# B&R Automation Studio project Parker_BMM_ST_V5_3147_V12 (part 14)

#### robot.c
```c
/********************************************************************
 * COPYRIGHT --  B&R
 ********************************************************************
 * Program: robot
 * File: robot.c
 * Author: lijianjun
 * Created: March 06, 2013
 ********************************************************************
 * Implementation of program robot --- robot control
 ********************************************************************/

#include <bur/plctypes.h>

#ifdef _DEFAULT_INCLUDES
#include <AsDefault.h>
#endif

/**************************************************************************************
                            Function Declarations
**************************************************************************************/
void RobotTransfer( Mold_typ * pMold,Robot_Para_typ * pRobotPara, Robot_Transfer_Fix_typ * pRobotTransferFix, Robot_UpDn_Fix_typ * pRobotUpDnFix );
void RobotTransfer_Drive( Mold_typ * pMold,Robot_Para_typ * pRobotPara, Robot_Transfer_Fix_typ * pRobotTransferFix, Robot_UpDn_Fix_typ * pRobotUpDnFix );

/**************************************************************************************
     	        		I N I T U P  O F   T H E   T A S K
**************************************************************************************/
_INIT void init ( void )
{
	RTInfo_Task.enable = 1;
	RTInfo(&RTInfo_Task);

	tTask = RTInfo_Task.cycle_time/1000.0/1000.0;		/*  from us ---> s  */

	LMold.Robot.Step = 30000;
	RMold.Robot.Step = 30000;

} /* end of _INIT */

 /*************************************************************************************
        				C Y C L I C   P A R T   O F   T H E   T A S K
**************************************************************************************/

_CYCLIC void cyclic ( void )
{
	if(LMold.TimeSet.RobotFwAlarmTime  == 0)LMold.TimeSet.RobotFwAlarmTime = 1000;	/*  10s  */
	if(LMold.TimeSet.RobotBwAlarmTime  == 0)LMold.TimeSet.RobotBwAlarmTime = 1000;
	if(LMold.TimeSet.RobotUpAlarmTime  == 0)LMold.TimeSet.RobotUpAlarmTime = 1000;
	if(LMold.TimeSet.RobotDnAlarmTime  == 0)LMold.TimeSet.RobotDnAlarmTime = 1000;

	if(RMold.TimeSet.RobotFwAlarmTime  == 0)RMold.TimeSet.RobotFwAlarmTime = 1000;	/*  10s  */
	if(RMold.TimeSet.RobotBwAlarmTime  == 0)RMold.TimeSet.RobotBwAlarmTime = 1000;
	if(RMold.TimeSet.RobotUpAlarmTime  == 0)RMold.TimeSet.RobotUpAlarmTime = 1000;
	if(RMold.TimeSet.RobotDnAlarmTime  == 0)RMold.TimeSet.RobotDnAlarmTime = 1000;

	LMold.TransDIn.RobotBwLimit = gMachineIn.LMold.RobotBwLimit;
	RMold.TransDIn.RobotBwLimit = gMachineIn.RMold.RobotBwLimit;

	LMold.TransDIn.RobotFwLimit = gMachineIn.LMold.RobotFwLimit;
	RMold.TransDIn.RobotFwLimit = gMachineIn.RMold.RobotFwLimit;

	LMold.TransDIn.RobotFwSlowLimit = gMachineIn.LMold.RobotFwSlowLimit;
	RMold.TransDIn.RobotFwSlowLimit = gMachineIn.RMold.RobotFwSlowLimit;

	LMold.TransDIn.RobotUpLimit = gMachineIn.LMold.RobotUpLimit;
	LMold.TransDIn.RobotDnLimit = gMachineIn.LMold.RobotDnLimit;

	RMold.TransDIn.RobotUpLimit = gMachineIn.RMold.RobotUpLimit;
	RMold.TransDIn.RobotDnLimit = gMachineIn.RMold.RobotDnLimit;

	//Ext Robot
	LMold.TransDIn.ExtRobotUpLmit = gMachineIn.LMold.ExtRobotUpLimit;
	RMold.TransDIn.ExtRobotUpLmit = gMachineIn.RMold.ExtRobotUpLimit;

	if(ACTUATOR_ELECTRIC == gMachineFix.MoldR.RobotTransfer.eActuatorType)
	{
		if(0 == gMachineFix.Option.bHideLeftStation)  // two mold
		{
			RobotTransfer_Drive(&LMold,&gMachinePara.MoldL.Robot,&gMachineFix.MoldL.RobotTransfer,&gMachineFix.MoldL.RobotUpDn);
		}
		RobotTransfer_Drive(&RMold,&gMachinePara.MoldR.Robot,&gMachineFix.MoldR.RobotTransfer,&gMachineFix.MoldR.RobotUpDn);
	}
	else
	{
		if(0 == gMachineFix.Option.bHideLeftStation)  // two mold
		{
			RobotTransfer(&LMold,&gMachinePara.MoldL.Robot,&gMachineFix.MoldL.RobotTransfer,&gMachineFix.MoldL.RobotUpDn);
		}
		RobotTransfer(&RMold,&gMachinePara.MoldR.Robot,&gMachineFix.MoldR.RobotTransfer,&gMachineFix.MoldR.RobotUpDn);
	}

	gMachineOut.LMold.RobotFw = LMold.ValveOut.RobotFw;
	gMachineOut.LMold.RobotBw = LMold.ValveOut.RobotBw;

	gMachineOut.RMold.RobotFw = RMold.ValveOut.RobotFw;
	gMachineOut.RMold.RobotBw = RMold.ValveOut.RobotBw;

	gMachineOut.LMold.RobotUp = LMold.ValveOut.RobotUp;
	gMachineOut.LMold.RobotDn = LMold.ValveOut.RobotDn;

	gMachineOut.RMold.RobotUp = RMold.ValveOut.RobotUp;
	gMachineOut.RMold.RobotDn = RMold.ValveOut.RobotDn;

	//		gMachineOut.LMold.ProductAuxClamp = LMold.ValveOut.ProductAuxClamp;
	//		gMachineOut.RMold.ProductAuxClamp = RMold.ValveOut.ProductAuxClamp;

	/*---------------------------------------------------*/
	/*----------------- Robot Transfer-----------------*/
	/*------------- ActuatorType--------------- */
	gMachineFix.MoldL.RobotTransfer.eActuatorType = gMachineFix.MoldR.RobotTransfer.eActuatorType;

	/*-------------- ValveType----------------- */
	gMachineFix.MoldL.RobotTransfer.eValveType = gMachineFix.MoldR.RobotTransfer.eValveType;

	/*------------ PressueOutputType--------------- */
	gMachineFix.MoldL.RobotTransfer.ePressueOutputType = gMachineFix.MoldR.RobotTransfer.ePressueOutputType;

	/*------------ FluxOutputType--------------- */
	gMachineFix.MoldL.RobotTransfer.eFluxOutputType = gMachineFix.MoldR.RobotTransfer.eFluxOutputType;

	/*---------------------------------------------------*/
	/*----------------- Robot UpDn-----------------*/
	/*------------- ActuatorType--------------- */
	gMachineFix.MoldL.RobotUpDn.eActuatorType = gMachineFix.MoldR.RobotUpDn.eActuatorType;

	/*-------------- ValveType----------------- */
	gMachineFix.MoldL.RobotUpDn.eValveType = gMachineFix.MoldR.RobotUpDn.eValveType;

	/*------------ PressueOutputType--------------- */
	gMachineFix.MoldL.RobotUpDn.ePressueOutputType = gMachineFix.MoldR.RobotUpDn.ePressueOutputType;

	/*------------ FluxOutputType--------------- */
	gMachineFix.MoldL.RobotUpDn.eFluxOutputType = gMachineFix.MoldR.RobotUpDn.eFluxOutputType;

	/*---------------Motor Trand-------------*/
	gMotorTrace.RMold.RobotTransfer.Position 		= RMold.Robot.Transfer.mmAs;

} /* end of _CYCLIC */

void RobotTransfer( Mold_typ * pMold,Robot_Para_typ * pRobotPara, Robot_Transfer_Fix_typ * pRobotTransferFix, Robot_UpDn_Fix_typ * pRobotUpDnFix )
{
	if(pMold == & LMold)
	{
		pRobotTransferFix->pMax = gMachineFix.Pump.MaxP2;
	}
	else
	{
		pRobotTransferFix->pMax = gMachineFix.Pump.MaxP1;
	}

	pMold->Robot.Transfer.FwPos = pMold->TransDIn.RobotFwLimit;
	pMold->Robot.Transfer.BwPos = pMold->TransDIn.RobotBwLimit;

	pMold->Robot.UpDn.UpPos = pMold->TransDIn.RobotUpLimit;
	pMold->Robot.UpDn.DnPos = pMold->TransDIn.RobotDnLimit;

	switch ( pMold->Robot.Step )
	{
		/*------------------ stop all the output ------------------*/
		case 0:

			switch (pRobotTransferFix->eActuatorType)
			{
				/*-------------------------------------------------*/
				case ACTUATOR_HYD: /*1:Oil*/
					/*-------------------------------------------------*/

					pMold->ActInfo.RobotFw	= 0;
					pMold->ActInfo.RobotBw	= 0;

					pMold->ValveOut.RobotFw = 0;
					pMold->ValveOut.RobotBw = 0;

					pMold->Robot.Transfer.p_set = 0;
					pMold->Robot.Transfer.v_set = 0;
					break;
				/*-------------------------------------------------*/
				case ACTUATOR_PNEU: /*2:Air*/
					/*-------------------------------------------------*/

					break;
			}

			pMold->Robot.Timer.IN = 0;
			pMold->Robot.LimitTimer.IN = 0;

			break;

		/*--------------------------------------------------- */
		/*------------------ Robot Fw ----------------------- */
		/*--------------------------------------------------- */
		case 100:		/* Fw delay */
			if(1 == pMold->Option.RobotTransfer)
			{
				if(pMold->TimeSet.RobotFwDly != 0)
				{
					pMold->Robot.Timer.IN = 1;
					pMold->Robot.Timer.PT = pMold->TimeSet.RobotFwDly;

					if(1 == gMachineInfo.Auto)
					{
						if(13000 == pMold->RobotOpnCls.Step || 0 == pMold->RobotOpnCls.Step)  // Opn too Slow wait, Opn Done
						{
							pMold->Robot.Step = 200;
						}
					}
					else
					{
						pMold->Robot.Step = 200;
					}
				}
				else
				{
					if(1 == gMachineInfo.Auto)
					{
						if(13000 == pMold->RobotOpnCls.Step || 0 == pMold->RobotOpnCls.Step)  // Opn too Slow wait, Opn Done
						{
							pMold->Robot.Step = 300;
						}
					}
					else
					{
						pMold->Robot.Step = 300;
					}
				}
			}
			else
			{
				pMold->Robot.Step = 300;
			}

			break;

		case 200:  		/* delay ok */
			pMold->TimeDis.RobotFwDly = pMold->Robot.Timer.ET;
			if (1 == pMold->Robot.Timer.Q)
			{
				pMold->Robot.Timer.IN        = 0;
				pMold->Robot.Step = 300;
			}
			break;

		case 300:  		/* set time */

			if(1 == pMold->Option.RobotTransfer)
			{
				pMold->Robot.LimitTimer.IN = 1;
				pMold->Robot.LimitTimer.PT = pMold->TimeSet.RobotFwAlarmTime;

				pMold->Robot.Step = 400;
			}
			else
			{
				pMold->Robot.Step = 2900; // for no use
			}
			break;

		case 400: // Fw quick
			pMold->ActInfo.RobotFw  = 1;
			pMold->ActInfo.RobotBw  = 0;

			switch (pRobotTransferFix->eActuatorType)
			{
				/*-------------------------------------------------*/
				case ACTUATOR_HYD: /*1:Oil*/
					/*-------------------------------------------------*/
					pMold->ValveOut.RobotFw = 1;
					pMold->ValveOut.RobotBw = 0;

					pMold->Robot.Transfer.p_set = pRobotPara->ParaTransfer.P_Fw;
					pMold->Robot.Transfer.v_set = pRobotPara->ParaTransfer.V_Fw;

					if(1 == pMold->TransDIn.RobotFwLimit || 1 == pMold->TransDIn.RobotFwSlowLimit)
					{
						pMold->Robot.Step = 500;
					}

					break;
				/*-------------------------------------------------*/
				case ACTUATOR_PNEU: /*2:Air*/
					/*-------------------------------------------------*/
					pMold->ValveOut.RobotFw = 1;
					pMold->ValveOut.RobotBw = 0;

					if(1 == pMold->TransDIn.RobotFwLimit )
					{
						pMold->Robot.Step = 1000;
					}

					break;
			}

			break;

		case 500: // Fw slow
			pMold->ActInfo.RobotFw  = 1;
			pMold->ActInfo.RobotBw  = 0;

			switch (pRobotTransferFix->eActuatorType)
			{
				/*-------------------------------------------------*/
				case ACTUATOR_HYD: /*1:Oil*/
					/*-------------------------------------------------*/
					pMold->ValveOut.RobotFw = 1;
					pMold->ValveOut.RobotBw = 0;

					pMold->Robot.Transfer.p_set = pRobotPara->ParaTransfer.P_FwSlow;
					pMold->Robot.Transfer.v_set = pRobotPara->ParaTransfer.V_FwSlow;

					if(1 == pMold->TransDIn.RobotFwLimit)
					{
						pMold->Robot.Timer.IN = 0;
						pMold->Robot.LimitTimer.IN   = 0;

						pMold->Robot.Step = 1000;
					}

					break;
				/*-------------------------------------------------*/
				case ACTUATOR_PNEU: /*2:Air*/
					/*-------------------------------------------------*/

					break;
			}

			break;

		case 1000:
			switch (pRobotTransferFix->eActuatorType)
			{
				/*-------------------------------------------------*/
				case ACTUATOR_HYD: /*1:Oil*/
					/*-------------------------------------------------*/
					pMold->ActInfo.RobotBw	= 0;
					pMold->ActInfo.RobotFw	= 0;

					pMold->ValveOut.RobotBw = 0;
					pMold->ValveOut.RobotFw = 0;

					pMold->Robot.Transfer.p_set = 0;
					pMold->Robot.Transfer.v_set = 0;

					pMold->Robot.Timer.IN = 0;
					pMold->Robot.LimitTimer.IN = 0;

					if(1 == gMachineInfo.Auto)
					{
						pMold->RobotOpnCls.Step = 100;  //Robot Cls
						pMold->Robot.Step = 2000;
					}
					else
					{
						pMold->Robot.Step = 3000;
					}

					break;
				/*-------------------------------------------------*/
				case ACTUATOR_PNEU: /*2:Air*/
					/*-------------------------------------------------*/
					pMold->ActInfo.RobotBw	= 0;
					pMold->ActInfo.RobotFw	= 1;

					pMold->ValveOut.RobotBw = 0;
					pMold->ValveOut.RobotFw = 1;

					pMold->Robot.Timer.IN = 0;
					pMold->Robot.LimitTimer.IN = 0;

					if(1 == gMachineInfo.Auto)
					{
						pMold->RobotOpnCls.Step = 100;  //Robot Cls
						pMold->Robot.Step = 2000;
					}
					else
					{
						pMold->Robot.Step = 3000;
					}

					break;
			}
			break;

		case 2000:  // wait  Robot Cls

			if( 3000 == pMold->RobotOpnCls.Step)
			{
				pMold->Robot.Step = 3000;
			}

			if( 40000 == pMold->RobotOpnCls.Step)
			{
				pMold->Robot.Step = 40000;
			}

			break;

		case 2900:  // for no use
			pMold->ActInfo.RobotBw	= 0;
			pMold->ActInfo.RobotFw	= 0;

			pMold->ValveOut.RobotBw = 0;
			pMold->ValveOut.RobotFw = 0;

			pMold->Robot.Transfer.p_set = 0;
			pMold->Robot.Transfer.v_set = 0;

			pMold->Robot.Timer.IN = 0;
			pMold->Robot.LimitTimer.IN = 0;

			if(1 == gMachineInfo.Auto)
			{
				pMold->RobotOpnCls.Step = 100;  //Robot Cls
			}

			pMold->Robot.Step = 3000;

			break;

		case 3000:
			break;

		/* ---------------------- calibration Fw ---------------------- */
		case 5000:
			pMold->ActInfo.RobotBw	= 0;
			pMold->ActInfo.RobotFw	= 1;

			pMold->ValveOut.RobotBw = 0;
			pMold->ValveOut.RobotFw = 1;

			pMold->Robot.Transfer.p_set = pRobotTransferFix->pCalibMax;
			pMold->Robot.Transfer.v_set = pRobotTransferFix->vCalibMax;

			break;

		/*--------------------------------------------------- */
		/*------------------ Robot Bw  ---------------------- */
		/*--------------------------------------------------- */
		case 10100:		/* Bw delay */
			if(1 == pMold->Option.RobotTransfer)
			{
				switch (pRobotTransferFix->eActuatorType)
				{
					/*-------------------------------------------------*/
					case ACTUATOR_HYD: /*1:Oil*/
						/*-------------------------------------------------*/
						if(pMold->TimeSet.RobotBwDly != 0)
						{
							pMold->Robot.Timer.IN = 1;
							pMold->Robot.Timer.PT = pMold->TimeSet.RobotBwDly;

							pMold->Robot.Step = 10200;
						}
						else
						{
							pMold->Robot.Step = 10300;
						}

						break;
					/*-------------------------------------------------*/
					case ACTUATOR_PNEU: /*2:Air*/
						/*-------------------------------------------------*/
						if(pMold->TimeSet.RobotBwDly != 0)
						{
							pMold->Robot.Timer.IN = 1;
							pMold->Robot.Timer.PT = pMold->TimeSet.RobotBwDly;

							pMold->Robot.Step = 10200;
						}
						else
						{
							pMold->Robot.Step = 10300;
						}

						break;
				}
			}
			else
			{
				pMold->Robot.Step = 10300;
			}

			break;

		case 10200:  		/* delay ok */
			pMold->TimeDis.RobotBwDly = pMold->Robot.Timer.ET;
			if (1 == pMold->Robot.Timer.Q)
			{
				pMold->Robot.Timer.IN  = 0;
				pMold->Robot.Step = 10300;
			}
			break;

		case 10300:
			if(pMold->Option.RobotTransfer)
			{
				pMold->Robot.LimitTimer.IN = 1;
				pMold->Robot.LimitTimer.PT = pMold->TimeSet.RobotBwAlarmTime;
				pMold->Robot.Step = 10400;
			}
			else  // for no use check limit
			{
				if (1 == pMold->Robot.Transfer.BwPos)
				{
					pMold->Robot.Step = 12900; // for no use
				}
				else
				{
					pMold->Alarm.RobotNotAtBwPos = !pMold->Robot.Transfer.BwPos;
					pMold->Robot.Step = 40000;     /*  Robot Bw alarm   */
				}
			}
			break;

		case 10400: // Bw quick
			pMold->ActInfo.RobotFw  = 0;
			pMold->ActInfo.RobotBw  = 1;

			switch (pRobotTransferFix->eActuatorType)
			{
				/*-------------------------------------------------*/
				case ACTUATOR_HYD: /*1:Oil*/
					/*-------------------------------------------------*/
					pMold->ValveOut.RobotFw = 0;
					pMold->ValveOut.RobotBw = 1;

					pMold->Robot.Transfer.p_set = pRobotPara->ParaTransfer.P_Bw;
					pMold->Robot.Transfer.v_set = pRobotPara->ParaTransfer.V_Bw;

					if(1 == pMold->TransDIn.RobotBwLimit || 1 == pMold->TransDIn.RobotBwSlowLimit)
					{
						pMold->Robot.Step = 10500;
					}

					break;
				/*-------------------------------------------------*/
				case ACTUATOR_PNEU: /*2:Air*/
					/*-------------------------------------------------*/
					pMold->ValveOut.RobotFw = 0;
					pMold->ValveOut.RobotBw = 1;

					if(1 == pMold->TransDIn.RobotBwLimit )
					{
						pMold->Robot.Step = 11000;
					}

					break;
			}

			break;

		case 10500: // Bw slow
			pMold->ActInfo.RobotFw  = 0;
			pMold->ActInfo.RobotBw  = 1;

			switch (pRobotTransferFix->eActuatorType)
			{
				/*-------------------------------------------------*/
				case ACTUATOR_HYD: /*1:Oil*/
					/*-------------------------------------------------*/
					pMold->ValveOut.RobotFw = 0;
					pMold->ValveOut.RobotBw = 1;

					pMold->Robot.Transfer.p_set = pRobotPara->ParaTransfer.P_BwSlow;
					pMold->Robot.Transfer.v_set = pRobotPara->ParaTransfer.V_BwSlow;

					if(1 == pMold->TransDIn.RobotBwLimit)
					{
						pMold->Robot.Timer.IN = 0;
						pMold->Robot.LimitTimer.IN   = 0;

						pMold->Robot.Step = 11000;
					}

					break;
				/*-------------------------------------------------*/
				case ACTUATOR_PNEU: /*2:Air*/
					/*-------------------------------------------------*/

					break;
			}

			break;

		case 11000:
			switch (pRobotTransferFix->eActuatorType)
			{
				/*-------------------------------------------------*/
				case ACTUATOR_HYD: /*1:Oil*/
					/*-------------------------------------------------*/
					pMold->ActInfo.RobotBw	= 0;
					pMold->ActInfo.RobotFw	= 0;

					pMold->ValveOut.RobotBw = 0;
					pMold->ValveOut.RobotFw = 0;

					pMold->Robot.Transfer.p_set = 0;
					pMold->Robot.Transfer.v_set = 0;

					pMold->Robot.Timer.IN = 0;
					pMold->Robot.LimitTimer.IN = 0;

					if(1 == gMachineInfo.Auto)
					{
						pMold->RobotOpnCls.Step = 10100;  //Robot Opn
						pMold->Robot.Step = 12000;

						if(0 == gMachineInfo.MachineReset)
						{
							pMold->CoolPin2.Step = 100;         /*  轉二下		 */
							pMold->CoolPin2Blow.Step =100;      /*  轉二下吹冷  */
							pMold->CoolPin3.Step = 100;	       	/*  轉三下		 */
							pMold->CoolPin3Blow.Step =100;    	/*  轉三下吹冷  */
						}
					}
					else
					{
						pMold->Robot.Step = 13000;
					}

					break;
				/*-------------------------------------------------*/
				case ACTUATOR_PNEU: /*2:Air*/
					/*-------------------------------------------------*/
					pMold->ActInfo.RobotBw	= 0;
					pMold->ActInfo.RobotFw	= 0;

					pMold->ValveOut.RobotBw = 0;
					pMold->ValveOut.RobotFw = 0;

					pMold->Robot.Timer.IN = 0;
					pMold->Robot.LimitTimer.IN = 0;

					if(1 == gMachineInfo.Auto)
					{
						pMold->RobotOpnCls.Step = 10100;  //Robot Opn
						pMold->Robot.Step = 12000;

						if(0 == gMachineInfo.MachineReset)
						{
							pMold->CoolPin2.Step = 100;         /*  轉二下		 */
							pMold->CoolPin2Blow.Step =100;      /*  轉二下吹冷  */
							pMold->CoolPin3.Step = 100;	       	/*  轉三下		 */
							pMold->CoolPin3Blow.Step =100;    	/*  轉三下吹冷  */
						}
					}
					else
					{
						pMold->Robot.Step = 13000;
					}

					break;
			}

			break;

		case 12000:  // wait Robot Opn

			if( 13000 == pMold->RobotOpnCls.Step)
			{
				pMold->RobotOpnCls.Step = 0;
				pMold->Robot.Step = 13000;
			}

			if( 40000 == pMold->RobotOpnCls.Step)
			{
				pMold->Robot.Step = 40000;
			}

			break;

		case 12900:  // for no use

			pMold->ActInfo.RobotBw	= 0;
			pMold->ActInfo.RobotFw	= 0;

			pMold->ValveOut.RobotBw = 0;
			pMold->ValveOut.RobotFw = 0;

			pMold->Robot.Transfer.p_set = 0;
			pMold->Robot.Transfer.v_set = 0;

			pMold->Robot.Timer.IN = 0;
			pMold->Robot.LimitTimer.IN = 0;

			if(1 == gMachineInfo.Auto)
			{
				pMold->RobotOpnCls.Step = 10100;  //Robot Opn
			}

			pMold->Robot.Step = 13000;

			break;

		case 13000:
			break;

		/* ---------------------- calibration Bw ---------------------- */
		case 15000:
			pMold->ActInfo.RobotFw	= 0;
			pMold->ActInfo.RobotBw	= 1;

			pMold->ValveOut.RobotFw = 0;
			pMold->ValveOut.RobotBw = 1;

			pMold->Robot.Transfer.p_set = pRobotTransferFix->pCalibZero;
			pMold->Robot.Transfer.v_set = pRobotTransferFix->vCalibZero;

			break;

		/* ------------- Normal stop ------------- */
		case 20000:
			switch (pRobotTransferFix->eActuatorType)
			{
				/*-------------------------------------------------*/
				case ACTUATOR_HYD: /*1:Oil*/
					/*-------------------------------------------------*/

					pMold->ActInfo.RobotFw	= 0;
					pMold->ActInfo.RobotBw	= 0;

					pMold->ValveOut.RobotFw = 0;
					pMold->ValveOut.RobotBw = 0;

					pMold->Robot.Transfer.p_set = 0;
					pMold->Robot.Transfer.v_set = 0;
					break;
				/*-------------------------------------------------*/
				case ACTUATOR_PNEU: /*2:Air*/
					/*-------------------------------------------------*/

					break;
			}

			pMold->Robot.Timer.IN = 0;
			pMold->Robot.LimitTimer.IN = 0;
			pMold->Robot.Step = 0;

			break;

		/* ------------- Instancy stop ------------- */
		case 30000:
			switch (pRobotTransferFix->eActuatorType)
			{
				/*-------------------------------------------------*/
				case ACTUATOR_HYD: /*1:Oil*/
					/*-------------------------------------------------*/

					pMold->ActInfo.RobotFw	= 0;
					pMold->ActInfo.RobotBw	= 0;

					pMold->ValveOut.RobotFw = 0;
					pMold->ValveOut.RobotBw = 0;

					pMold->Robot.Transfer.p_set = 0;
					pMold->Robot.Transfer.v_set = 0;
					break;
				/*-------------------------------------------------*/
				case ACTUATOR_PNEU: /*2:Air*/
					/*-------------------------------------------------*/

					break;
			}

			pMold->Robot.Timer.IN = 0;
			pMold->Robot.LimitTimer.IN = 0;
			pMold->Robot.Step = 0;

			break;

		/* ------------- Error stop ------------- */
		case 40000:
			switch (pRobotTransferFix->eActuatorType)
			{
				/*-------------------------------------------------*/
				case ACTUATOR_HYD: /*1:Oil*/
					/*-------------------------------------------------*/

					pMold->ActInfo.RobotFw	= 0;
					pMold->ActInfo.RobotBw	= 0;

					pMold->ValveOut.RobotFw = 0;
					pMold->ValveOut.RobotBw = 0;

					pMold->Robot.Transfer.p_set = 0;
					pMold->Robot.Transfer.v_set = 0;
					break;
				/*-------------------------------------------------*/
				case ACTUATOR_PNEU: /*2:Air*/
					/*-------------------------------------------------*/

					break;
			}

			pMold->Robot.Timer.IN = 0;
			pMold->Robot.LimitTimer.IN = 0;
			pMold->Robot.Step = 0;

			break;

		/* ------------- auto run stop ------------- */
		case 41000:
			switch (pRobotTransferFix->eActuatorType)
			{
				/*-------------------------------------------------*/
				case ACTUATOR_HYD: /*1:Oil*/
					/*-------------------------------------------------*/

					pMold->ActInfo.RobotFw	= 0;
					pMold->ActInfo.RobotBw	= 0;

					pMold->ValveOut.RobotFw = 0;
					pMold->ValveOut.RobotBw = 0;

					pMold->Robot.Transfer.p_set = 0;
					pMold->Robot.Transfer.v_set = 0;
					break;
				/*-------------------------------------------------*/
				case ACTUATOR_PNEU: /*2:Air*/
					/*-------------------------------------------------*/

					break;
			}

			pMold->Robot.Timer.IN = 0;
			pMold->Robot.LimitTimer.IN = 0;
			pMold->Robot.Step = 40000;

			break;
	}/* end of switch */

	/* ----------------- Robot Fw/Bw alarm time display --------------------  */
	if(pMold->Robot.Step > 300 && pMold->Robot.Step  < 1000)			/* Robot Fw  */
	{
		pMold->TimeDis.RobotFwAlarmTime = pMold->Robot.LimitTimer.ET;
	}
	else if(pMold->Robot.Step > 10300 && pMold->Robot.Step  < 11000)	/* Robot Bw   */
	{
		pMold->TimeDis.RobotBwAlarmTime = pMold->Robot.LimitTimer.ET;
	}

	/* ----------------- Robot Fw/Bw timeout --------------------  */
	if(1 == pMold->Robot.LimitTimer.Q  && 1 == gMachineInfo.TimeLimit)
	{
		if(pMold->Robot.Step < 3000 && pMold->Robot.Step > 200)		/* Robot Fw  */
		{
			pMold->Alarm.RobotNotAtFwPos = 1;
		}

		if(pMold->Robot.Step < 13000 && pMold->Robot.Step > 10200)	/* Robot Bw   */
		{
			pMold->Alarm.RobotNotAtBwPos = 1;
		}

		pMold->Robot.Step = 41000;
	}/* if(1 == pMold->Robot.LimitTimer.Q) */

	/* ----------------- Robot Fw/Bw action limit --------------------  */
	if(pMold->Robot.Step < 3000 && pMold->Robot.Step > 200)		/* Robot Fw  */
	{
		if(0 == pMold->Carriage.BwPos)
		{
			pMold->Alarm.CarriageNotAtBwDI = !pMold->Carriage.BwPos;
			pMold->Robot.Step = 40000;
		}

		if(0 == gMachineInfo.Auto || (1 == gMachineInfo.Auto && 1 == gMachineFix.Option.bRobotFwAfterTopdeflash))
		{
			if( 0 == pMold->TransDIn.TopDeflashBwLimit )
			{
				pMold->Alarm.TopDeflashNotAtBwPos = !pMold->TransDIn.TopDeflashBwLimit;
				pMold->Robot.Step = 41000;
			}
		}

		if( 0 == pMold->TransDIn.RobotOpnLimit)
		{
			pMold->Alarm.RobotNotAtOpnPos = !pMold->TransDIn.RobotOpnLimit;
			pMold->Robot.Step = 41000;
		}

	}

	if(pMold->Robot.Step < 13000 && pMold->Robot.Step > 10200)	/* Robot Bw   */
	{
		if(0 == gMachineInfo.Auto)
		{
			if(0 == pMold->Clamp.OpnPos)
			{
				pMold->Alarm.ClampNotAtOpnDI = !pMold->Clamp.OpnPos;
				pMold->Robot.Step = 41000;
			}
		}
		else if(1 == gMachineInfo.Auto)
		{
			if(0 == (pMold->Clamp.mmAs > (pMold->Clamp.S_OpnEnd - pMold->Clamp.Tolerance)) && 0 == pMold->Carriage.FwPos )
			{
				pMold->Alarm.ClampNotAtOpnDI = !(pMold->Clamp.mmAs > (pMold->Clamp.S_OpnEnd - pMold->Clamp.Tolerance));
				pMold->Alarm.CarriageNotAtFwDI = !pMold->Carriage.FwPos;
				pMold->Robot.Step = 41000;
			}
		}

		if( 0 == pMold->TransDIn.CoolPinUpLimit)
		{
			pMold->Alarm.CoolPinNotAtUpPos  = !pMold->TransDIn.CoolPinUpLimit;
			pMold->Robot.Step = 41000;
		}

		if(0 == pMold->TransDIn.CoolPin2UpLimit)
		{
			pMold->Alarm.CoolPin2NotAtUpPos = !pMold->TransDIn.CoolPin2UpLimit;
			pMold->Robot.Step = 41000;
		}

		if(0 == pMold->TransDIn.CoolPin3UpLimit)
		{
			pMold->Alarm.CoolPin3NotAtUpPos = !pMold->TransDIn.CoolPin3UpLimit;
			pMold->Robot.Step = 41000;
		}

	}

}/*end of function */

void RobotTransfer_Drive( Mold_typ * pMold,Robot_Para_typ * pRobotPara, Robot_Transfer_Fix_typ * pRobotTransferFix, Robot_UpDn_Fix_typ * pRobotUpDnFix )
{
	if(pMold == & LMold)
	{
		pRobotTransferFix->pMax = 100;
	}
	else
	{
		pRobotTransferFix->pMax = 100;
	}

	if(1 == gMachineOut.OilPump)
	{
		if(tErrorDelay >= tTask)tErrorDelay = tErrorDelay - tTask;
		if(tErrorDelay < tTask)
		{
			if(pMold == & LMold)
			{
				LMold.HwAlarm.RobotTransferAxisErr = !LMold.Robot.Transfer.NetworkInit;
				LMold.HwAlarm.RobotTransferPowerOn = !LMold.Robot.Transfer.PowerOn;
			}
			else
			{
				RMold.HwAlarm.RobotTransferAxisErr = !RMold.Robot.Transfer.NetworkInit;
				RMold.HwAlarm.RobotTransferPowerOn = !RMold.Robot.Transfer.PowerOn;
			}
		}

		if((RMold.HwAlarm.RobotTransferAxisErr ||RMold.HwAlarm.RobotTransferPowerOn)||(LMold.HwAlarm.RobotTransferAxisErr ||LMold.HwAlarm.RobotTransferPowerOn))
		{
			gMachineOut.OilPump = 0;
			gPROCESS_info.oilpumpStop = 1;   //request manual mode
		}
	}
	else
	{
		tErrorDelay = 0.1;
		if(pMold == & LMold)
		{
			//			LMold.HwAlarm.RobotTransferPowerOn = 0;
			//			LMold.HwAlarm.RobotTransferPowerOn = 0;
		}
		else
		{
			//			RMold.HwAlarm.RobotTransferPowerOn = 0;
			//			RMold.HwAlarm.RobotTransferPowerOn = 0;
		}
	}

	/* ------------- robot transfer axis alarms ------------- */

	pMold->HwAlarm.RobotTransferAxisErr    = pMold->Robot.Transfer.Error;

	/*********************************************************************************
  	**                            HMI data value to PLC                             **
  	*********************************************************************************/
	if(pRobotTransferFix->Tolerance < 0.3)pRobotTransferFix->Tolerance = 2.0;
	if(0 == pRobotPara->ParaTransfer.V_BwReset)pRobotPara->ParaTransfer.V_BwReset = 2.0;

	if(0 == pMold->Robot.Transfer.Error && 1 == pMold->Robot.Transfer.HomingOk && pRobotTransferFix->sHome != 0 &&
		pMold->Robot.Transfer.mmAs > -15 && pMold->Robot.Transfer.mmAs < pRobotTransferFix->sMax + 15)
	{
		pMold->Robot.Transfer.CalOK = 1;
	}
	else
	{
		pMold->Robot.Transfer.CalOK = 0;
	}

	//	if(0 == pMold->Robot.UpDn.Error && 1 == pMold->Robot.UpDn.HomingOk && pRobotUpDnFix->sHome != 0 &&
	//		pMold->Robot.UpDn.mmAs > -15 && pMold->Robot.UpDn.mmAs < pRobotUpDnFix->sMax + 15)
	//	{
	//		pMold->Robot.UpDn.CalOK = 1;
	//	}
	//	else
	//	{
	//		pMold->Robot.UpDn.CalOK = 0;
	//	}

	if(1 == pMold->Robot.Transfer.CalOK)
	{
		pMold->Robot.Transfer.BwPos = pMold->TransDIn.RobotBwLimit & (pMold->Robot.Transfer.mmAs <= pRobotPara->ParaTransfer.S_Bw + pRobotTransferFix->Tolerance) &
			(pMold->Robot.Transfer.mmAs >= pRobotPara->ParaTransfer.S_Bw - pRobotTransferFix->Tolerance);
		pMold->Robot.Transfer.FwPos = pMold->TransDIn.RobotFwLimit & (pMold->Robot.Transfer.mmAs >= pRobotPara->ParaTransfer.S_Fw - pRobotTransferFix->Tolerance) &
			(pMold->Robot.Transfer.mmAs <= pRobotPara->ParaTransfer.S_Fw + pRobotTransferFix->Tolerance);

		pMold->Robot.Transfer.WastePos = (pMold->Robot.Transfer.mmAs > pRobotPara->ParaTransfer.S_WasteFw - pRobotTransferFix->Tolerance) &
			(pMold->Robot.Transfer.mmAs < pRobotPara->ParaTransfer.S_WasteFw + pRobotTransferFix->Tolerance);

	}
	else
	{
		pMold->Robot.Transfer.BwPos = 0;
		pMold->Robot.Transfer.FwPos = 0;
		pMold->Robot.Transfer.WastePos = 0;
	}

	//	pRobotUpDnFix->Tolerance = 0.3;
	//
	//	if(1 == pMold->Robot.UpDn.CalOK)
	//	{
	//		pMold->Robot.UpDn.UpPos = pMold->TransDIn.RobotUpLimit & (pMold->Robot.UpDn.mmAs <= pRobotPara->ParaUpDn.sUp + pRobotUpDnFix->Tolerance) &
	//			(pMold->Robot.UpDn.mmAs >= pRobotPara->ParaUpDn.sUp - pRobotUpDnFix->Tolerance);
	//	}
	//	else
	//	{
	//		pMold->Robot.UpDn.UpPos = 0;
	//	}

	if(0 == pMold->Robot.Transfer.CalOK )
	{
		if(0 == gMachineInfo.Calib)	/* 非调校模式  */
		{
			if(pMold->Robot.Step > 0 && pMold->Robot.Step < 20000)
			{
				pMold->Alarm.RobotTransferCalErr = ! pMold->Robot.Transfer.CalOK;
				pMold->Robot.Step = 20000;
			}
		}
	}

	//	if(1 == pMold->Option.RobotUpDn && 0 == pMold->Robot.UpDn.CalOK)
	//	{
	//		if(0 == gMachineInfo.Calib)	/* 非调校模式  */
	//		{
	//			if(pMold->Robot.Step > 0 && pMold->Robot.Step < 20000)
	//			{
	//				pMold->Alarm.RobotUpDnCalErr = ! pMold->Robot.UpDn.CalOK;
	//				pMold->Robot.Step = 20000;
	//			}
	//		}
	//	}

	switch(pMold->Robot.Step)
	{
		case 0:
			pMold->Robot.Transfer.MoveAbsolute = 0;
			pMold->Robot.Transfer.MoveJogPos = 0;
			pMold->Robot.Transfer.MoveJogNeg = 0;
			pMold->Robot.Transfer.Stop = 0;

			pMold->Robot.UpDn.MoveAbsolute = 0;
			pMold->Robot.UpDn.MoveJogPos = 0;
			pMold->Robot.UpDn.MoveJogNeg = 0;
			pMold->Robot.UpDn.Stop = 0;

			pMold->ActInfo.RobotFw	= 0;
			pMold->ActInfo.RobotBw	= 0;
			pMold->ActInfo.RobotUp	= 0;
			pMold->ActInfo.RobotDn	= 0;

			pMold->Robot.Timer.IN = 0;
			pMold->Robot.LimitTimer.IN = 0;

			break;

		/*------------------------------------------------------- */
		/*---------------------- Robot Fw ----------------------- */
		/*------------------------------------------------------- */
		case 100:		/* fw delay */
			if(1 == pMold->Option.RobotTransfer)
			{
				if(pMold->TimeSet.RobotFwDly != 0)
				{
					pMold->Robot.Timer.IN = 1;
					pMold->Robot.Timer.PT = pMold->TimeSet.RobotFwDly;

					if(1 == gMachineInfo.Auto)
					{
						if(13000 == pMold->RobotOpnCls.Step || 0 == pMold->RobotOpnCls.Step)  // Opn too Slow wait, Opn Done
						{
							pMold->Robot.Step = 200;
						}
					}
					else
					{
						pMold->Robot.Step = 200;
					}
				}
				else
				{
					if(1 == gMachineInfo.Auto)
					{
						if(13000 == pMold->RobotOpnCls.Step || 0 == pMold->RobotOpnCls.Step)  // Opn too Slow wait, Opn Done
						{
							pMold->Robot.Step = 300;
						}
					}
					else
					{
						pMold->Robot.Step = 300;
					}
				}
			}
			else
			{
				pMold->Robot.Step = 300; // for no use
			}
			break;

		case 200:  		/* delay ok */
			pMold->TimeDis.RobotFwDly = pMold->Robot.Timer.ET;
			if (1 == pMold->Robot.Timer.Q)
			{
				pMold->Robot.Timer.IN        = 0;

				pMold->Robot.Step = 300;
			}
			break;

		case 300:		/* time limit  */

			if(1 == pMold->Option.RobotTransfer)
			{
				pMold->Robot.Transfer.MoveAbsolute = 1;
				pMold->Robot.Transfer.v_set = pRobotPara->ParaTransfer.V_Fw;
				pMold->Robot.Transfer.s_set = pRobotPara->ParaTransfer.S_Fw;

				pMold->Robot.LimitTimer.IN = 1;
				pMold->Robot.LimitTimer.PT = pMold->TimeSet.RobotFwAlarmTime;
				pMold->Robot.Step = 400;
			}
			else
			{
				pMold->Robot.Step = 2900; // for no use
			}

			if(1 == pMold->Robot.Transfer.FwHWSwitch)
			{
				pMold->HwAlarm.RobotTransferFwHWSwitch = 1;
				pMold->Robot.Step = 40000;
			}
			break;

		case 400:
			pMold->ActInfo.RobotFw  = 1;
			pMold->ActInfo.RobotBw  = 0;

			if(pMold->Robot.Transfer.mmAs >= pRobotPara->ParaTransfer.S_Fw - pRobotTransferFix->Tolerance) 	/*  機械手進位置到  */
			{
				pMold->Robot.Timer.IN = 0;
				pMold->Robot.LimitTimer.IN = 0;

				pMold->Robot.Step = 500;
			}

			if(1 == pMold->Robot.Transfer.FwHWSwitch)
			{
				pMold->HwAlarm.RobotTransferFwHWSwitch = 1;
				pMold->Robot.Step = 40000;
			}

			break;

		case 500:
			pMold->ActInfo.RobotFw	= 0;
			pMold->ActInfo.RobotBw	= 0;

			pMold->Robot.Transfer.MoveAbsolute = 0;
			pMold->Robot.Transfer.Stop = 1;

			pMold->Robot.Timer.IN   = 0;
			pMold->Robot.LimitTimer.IN = 0;

			if(1 == gMachineInfo.Auto)
			{
				pMold->RobotOpnCls.Step = 100;  //Robot Cls
			}

			pMold->Robot.Step = 3000;

			break;

		case 2900:	// for no use
			pMold->ActInfo.RobotFw	= 0;
			pMold->ActInfo.RobotBw	= 0;

			pMold->Robot.Transfer.MoveAbsolute = 0;
			pMold->Robot.Transfer.Stop = 1;

			pMold->Robot.Timer.IN   = 0;
			pMold->Robot.LimitTimer.IN = 0;

			if(1 == gMachineInfo.Auto)
			{
				pMold->RobotOpnCls.Step = 100;  //Robot Cls
			}

			pMold->Robot.Step = 3000;

			break;

		case 3000:
			break;

		/* ---------------------- calibration forward ---------------------- */
		case 5000:
			pMold->ActInfo.RobotFw  = 1;
			pMold->ActInfo.RobotBw  = 0;

			pMold->Robot.Transfer.v_set = pRobotTransferFix->vCalibMax;
			pMold->Robot.Transfer.MoveJogPos = 1;

			if(1 == pMold->Robot.Transfer.FwHWSwitch)
			{
				pMold->HwAlarm.RobotTransferFwHWSwitch = 1;
				pMold->Robot.Step = 40000;
			}

			break;

		/* ---------------------- calibration down ---------------------- */
		//		case 5500:
		//			pMold->Robot.UpDn.MoveJogPos = 1;
		//			if(1 == pMold->TransDIn.RobotDnLimit)
		//			{
		//				pMold->Robot.Step = 20000;
		//			}
		//			break;

		/*------------------------------------------------------- */
		/*---------------------- Robot Bw ----------------------- */
		/*------------------------------------------------------- */
		case 10100:		/* bw delay */
			if(1 == pMold->Option.RobotTransfer)
			{
				if(pMold->TimeSet.RobotBwDly != 0)
				{
					pMold->Robot.Timer.IN = 1;
					pMold->Robot.Timer.PT = pMold->TimeSet.RobotBwDly;

					pMold->Robot.Step = 10200;
				}
				else
				{
					pMold->Robot.Step = 10300;
				}
			}
			else
			{
				pMold->Robot.Step = 10300;
			}
			break;

		case 10200:  		/* delay ok */
			pMold->TimeDis.RobotBwDly = pMold->Robot.Timer.ET;
			if (1 == pMold->Robot.Timer.Q)
			{
				pMold->Robot.Timer.IN   = 0;
				pMold->Robot.Step = 10300;
			}
			break;

		case 10300:		/* time limit  */

			if(1 == pMold->Option.RobotTransfer)
			{
				pMold->Robot.Transfer.MoveAbsolute = 1;

				if(1 == gMachineInfo.MachineReset )
				{
					pMold->Robot.Transfer.v_set = pRobotPara->ParaTransfer.V_BwReset;
				}
				else
				{
					pMold->Robot.Transfer.v_set = pRobotPara->ParaTransfer.V_Bw;
				}
				pMold->Robot.Transfer.s_set = pRobotPara->ParaTransfer.S_Bw;
				pMold->Robot.LimitTimer.IN = 1;
				pMold->Robot.LimitTimer.PT = pMold->TimeSet.RobotBwAlarmTime;
				pMold->Robot.Step = 10400;
			}
			else   // for no use check limit
			{
				if (1 == pMold->Robot.Transfer.BwPos)
				{
					pMold->Robot.Step = 12900; // for no use
				}
				else
				{
					pMold->Alarm.RobotNotAtBwPos = !pMold->Robot.Transfer.BwPos;
					pMold->Robot.Step = 40000;
				}
			}

			if(1 == pMold->Robot.Transfer.BwHWSwitch)
			{
				pMold->HwAlarm.RobotTransferBwHWSwitch = 1;
				pMold->Robot.Step = 40000;
			}

			break;

		case 10400:
			pMold->ActInfo.RobotFw  = 0;
			pMold->ActInfo.RobotBw  = 1;

			if(pMold->Robot.Transfer.mmAs <= pRobotPara->ParaTransfer.S_Bw + pRobotTransferFix->Tolerance) 	/*  機械手退位置到  */
			{
				pMold->Robot.Timer.IN = 0;
				pMold->Robot.LimitTimer.IN = 0;

				pMold->Robot.Step = 10500;
			}

			if(1 == pMold->Robot.Transfer.BwHWSwitch)
			{
				pMold->HwAlarm.RobotTransferBwHWSwitch = 1;
				pMold->Robot.Step = 40000;
			}

			break;

		case 10500:
			pMold->ActInfo.RobotFw	= 0;
			pMold->ActInfo.RobotBw	= 0;

			pMold->Robot.Transfer.MoveAbsolute = 0;
			pMold->Robot.Transfer.Stop = 1;

			pMold->Robot.Timer.IN   = 0;
			pMold->Robot.LimitTimer.IN = 0;

			if(1 == gMachineInfo.Auto)
			{
				pMold->RobotOpnCls.Step = 10100;  //Robot Opn

				if(0 == gMachineInfo.MachineReset)
				{
					pMold->CoolPin2.Step = 100;         /*  轉二下		 */
					pMold->CoolPin2Blow.Step =100;      /*  轉二下吹冷  */
					pMold->CoolPin3.Step = 100;	       	/*  轉三下		 */
					pMold->CoolPin3Blow.Step =100;    	/*  轉三下吹冷  */
				}
			}
			pMold->Robot.Step = 13000;

			break;

		case 12900:  // for no use

			pMold->ActInfo.RobotFw	= 0;
			pMold->ActInfo.RobotBw	= 0;

			pMold->Robot.Transfer.MoveAbsolute = 0;
			pMold->Robot.Transfer.Stop = 1;

			pMold->Robot.Timer.IN   = 0;
			pMold->Robot.LimitTimer.IN = 0;

			if(1 == gMachineInfo.Auto)
			{
				pMold->RobotOpnCls.Step = 10100;  //Robot Opn
			}

			pMold->Robot.Step = 13000;

			break;

		case 13000:

			break;

		/* ---------------------- calibration backward ---------------------- */
		case 15000:
			pMold->ActInfo.RobotFw  = 0;
			pMold->ActInfo.RobotBw  = 1;

			pMold->Robot.Transfer.v_set = pRobotTransferFix->vCalibZero;
			pMold->Robot.Transfer.MoveJogNeg = 1;

			if(1 == pMold->Robot.Transfer.BwHWSwitch)
			{
				pMold->HwAlarm.RobotTransferBwHWSwitch = 1;
				pMold->Robot.Step = 40000;
			}
			break;

		/* ---------------------- calibration upward ---------------------- */
		//		case 15500:
		//			pMold->Robot.UpDn.MoveJogNeg = 1;
		//			break;

		/* ------------- Normal stop ------------- */
		case 20000:
			pMold->ActInfo.RobotFw  = 0;
			pMold->ActInfo.RobotBw  = 0;

			pMold->Robot.Transfer.MoveAbsolute = 0;
			pMold->Robot.Transfer.MoveJogPos = 0;
			pMold->Robot.Transfer.MoveJogNeg = 0;
			pMold->Robot.Transfer.Stop = 1;

			//			pMold->Robot.UpDn.MoveAbsolute = 0;
			//			pMold->Robot.UpDn.MoveJogPos = 0;
			//			pMold->Robot.UpDn.MoveJogNeg = 0;
			//			pMold->Robot.UpDn.Stop = 1;

			pMold->ActInfo.RobotFw	= 0;
			pMold->ActInfo.RobotBw	= 0;
			pMold->ActInfo.RobotUp	= 0;
			pMold->ActInfo.RobotDn	= 0;

			pMold->Robot.Timer.IN = 0;
			pMold->Robot.LimitTimer.IN = 0;

			pMold->Robot.Step = 0;
			break;

		/* ------------- Calib stop ------------- */
		case 25000:
			pMold->ActInfo.RobotFw  = 0;
			pMold->ActInfo.RobotBw  = 0;

			//			pMold->Robot.Transfer.MoveAbsolute = 0;
			pMold->Robot.Transfer.MoveJogPos = 0;
			pMold->Robot.Transfer.MoveJogNeg = 0;
			//			pMold->Robot.Transfer.Stop = 1;

			//			pMold->Robot.UpDn.MoveAbsolute = 0;
			//			pMold->Robot.UpDn.MoveJogPos = 0;
			//			pMold->Robot.UpDn.MoveJogNeg = 0;
			//			pMold->Robot.UpDn.Stop = 1;

			pMold->ActInfo.RobotFw	= 0;
			pMold->ActInfo.RobotBw	= 0;
			pMold->ActInfo.RobotUp	= 0;
			pMold->ActInfo.RobotDn	= 0;

			pMold->Robot.Timer.IN = 0;
			pMold->Robot.LimitTimer.IN = 0;

			pMold->Robot.Step = 0;
			break;

		/* ------------- Instancy stop ------------- */
		case 30000:
			pMold->Robot.Transfer.MoveAbsolute = 0;
			pMold->Robot.Transfer.MoveJogPos = 0;
			pMold->Robot.Transfer.MoveJogNeg = 0;
			pMold->Robot.Transfer.Stop = 1;

			//			pMold->Robot.UpDn.MoveAbsolute = 0;
			//			pMold->Robot.UpDn.MoveJogPos = 0;
			//			pMold->Robot.UpDn.MoveJogNeg = 0;
			//			pMold->Robot.UpDn.Stop = 1;

			pMold->ActInfo.RobotFw	= 0;
			pMold->ActInfo.RobotBw	= 0;
			//			pMold->ActInfo.RobotUp	= 0;
			//			pMold->ActInfo.RobotDn	= 0;

			pMold->Robot.Timer.IN = 0;
			pMold->Robot.LimitTimer.IN = 0;

			pMold->Robot.Step = 0;
			break;

		/* ------------- Error stop ------------- */
		case 40000:
			pMold->Robot.Transfer.MoveAbsolute = 0;
			pMold->Robot.Transfer.MoveJogPos = 0;
			pMold->Robot.Transfer.MoveJogNeg = 0;
			pMold->Robot.Transfer.Stop = 1;

			//			pMold->Robot.UpDn.MoveAbsolute = 0;
			//			pMold->Robot.UpDn.MoveJogPos = 0;
			//			pMold->Robot.UpDn.MoveJogNeg = 0;
			//			pMold->Robot.UpDn.Stop = 1;

			pMold->ActInfo.RobotFw	= 0;
			pMold->ActInfo.RobotBw	= 0;
			pMold->ActInfo.RobotUp	= 0;
			pMold->ActInfo.RobotDn	= 0;

			pMold->Robot.Timer.IN = 0;
			pMold->Robot.LimitTimer.IN = 0;

			//			gImply.RobotReset = 1;
			break;

		/* ------------- auto run stop ------------- */
		case 41000:
			pMold->Robot.Transfer.MoveAbsolute = 0;
			pMold->Robot.Transfer.MoveJogPos = 0;
			pMold->Robot.Transfer.MoveJogNeg = 0;
			pMold->Robot.Transfer.Stop = 1;

			//			pMold->Robot.UpDn.MoveAbsolute = 0;
			//			pMold->Robot.UpDn.MoveJogPos = 0;
			//			pMold->Robot.UpDn.MoveJogNeg = 0;
			//			pMold->Robot.UpDn.Stop = 1;

			pMold->ActInfo.RobotFw	= 0;
			pMold->ActInfo.RobotBw	= 0;
			//			pMold->ActInfo.RobotUp	= 0;
			//			pMold->ActInfo.RobotDn	= 0;

			pMold->Robot.Timer.IN = 0;
			pMold->Robot.LimitTimer.IN = 0;

			pMold->Robot.Step = 40000;
			break;
	}/* switch(pMold->Robot.Step) */

	/* ----------------- Robot Fw/Bw alarm time display --------------------  */
	if(pMold->Robot.Step > 300 && pMold->Robot.Step  < 1000)			/* Robot Fw  */
	{
		pMold->TimeDis.RobotFwAlarmTime = pMold->Robot.LimitTimer.ET;
	}
	else if(pMold->Robot.Step > 10300 && pMold->Robot.Step  < 11000)	/* Robot Bw   */
	{
		pMold->TimeDis.RobotBwAlarmTime = pMold->Robot.LimitTimer.ET;
	}

	/* ----------------- Robot Fw/Bw timeout --------------------  */
	if(1 == pMold->Robot.LimitTimer.Q  && 1 == gMachineInfo.TimeLimit)
	{
		if(pMold->Robot.Step < 3000 && pMold->Robot.Step > 200)		/* Robot Fw  */
		{
			pMold->Alarm.RobotNotAtFwPos = 1;
		}

		if(pMold->Robot.Step < 13000 && pMold->Robot.Step > 10200)	/* Robot Bw   */
		{
			pMold->Alarm.RobotNotAtBwPos = 1;
		}

		pMold->Robot.Step = 41000;
	}/* if(1 == pMold->Robot.LimitTimer.Q) */

	/* ----------------- Robot Fw/Bw action limit --------------------  */
	if(pMold->Robot.Step < 3000 && pMold->Robot.Step > 200)		/* Robot Fw  */
	{
		if(0 == pMold->Carriage.BwPos)
		{
			pMold->Alarm.CarriageNotAtBwDI = !pMold->Carriage.BwPos;
			pMold->Robot.Step = 40000;
		}

		if(0 == gMachineInfo.Auto || (1 == gMachineInfo.Auto && 1 == gMachineFix.Option.bRobotFwAfterTopdeflash))
		{
			if( 0 == pMold->TransDIn.TopDeflashBwLimit )
			{
				pMold->Alarm.TopDeflashNotAtBwPos = !pMold->TransDIn.TopDeflashBwLimit;
				pMold->Robot.Step = 41000;
			}
		}

		if( 0 == pMold->TransDIn.RobotOpnLimit)
		{
			pMold->Alarm.RobotNotAtOpnPos = !pMold->TransDIn.RobotOpnLimit;
			pMold->Robot.Step = 41000;
		}

	}

	if(pMold->Robot.Step < 13000 && pMold->Robot.Step > 10200)	/* Robot Bw   */
	{
		if(0 == gMachineInfo.Auto)
		{
			if(0 == pMold->Clamp.OpnPos)
			{
				pMold->Alarm.ClampNotAtOpnDI = !pMold->Clamp.OpnPos;
				pMold->Robot.Step = 41000;
			}
		}
		else if(1 == gMachineInfo.Auto)
		{
			//			if(0 == (pMold->Clamp.mmAs > (pMold->Clamp.S_OpnEnd - pMold->Clamp.Tolerance)) && 0 == pMold->Carriage.FwPos )
			//			{
			//				pMold->Alarm.ClampNotAtOpnDI = !(pMold->Clamp.mmAs > (pMold->Clamp.S_OpnEnd - pMold->Clamp.Tolerance));
			//				pMold->Alarm.CarriageNotAtFwDI = !pMold->Carriage.FwPos;
			//				pMold->Robot.Step = 41000;
			//			}

			if(0 == pMold->Clamp.OpnPos && 0 == pMold->Carriage.FwPos )
			{
				pMold->Alarm.ClampNotAtOpnDI = !pMold->Clamp.OpnPos;
				pMold->Alarm.CarriageNotAtFwDI = !pMold->Carriage.FwPos;
				pMold->Robot.Step = 41000;
			}
		}

		if(0 == pMold->TransDIn.CoolPin2UpLimit)
		{
			pMold->Alarm.CoolPin2NotAtUpPos = !pMold->TransDIn.CoolPin2UpLimit;
			pMold->Robot.Step = 41000;
		}

		if(0 == pMold->TransDIn.CoolPin3UpLimit)
		{
			pMold->Alarm.CoolPin3NotAtUpPos = !pMold->TransDIn.CoolPin3UpLimit;
			pMold->Robot.Step = 41000;
		}

	}

}/* void Robot(Mold_typ * pMold) */
```

#### robot.var
```iecst
VAR
	tTask : REAL := 0.0;
	RTInfo_Task : RTInfo := (0);
	tErrorDelay : REAL;
END_VAR
```

### Program Logical/process/robotopncls (ANSIC, version 1.00.0) - robot open /close

#### robotopncls.c
```c
/********************************************************************
 * COPYRIGHT --  B&R
 ********************************************************************
 * Program: robotopncls
 * File: robotopncls.c
 * Author: lijianjun
 * Created: March 06, 2013
 ********************************************************************
 * Implementation of program coolpin --- cooling pin control
 ********************************************************************/

#include <bur/plctypes.h>

#ifdef _DEFAULT_INCLUDES
#include <AsDefault.h>
#endif

/**************************************************************************************
                            Function Declarations
**************************************************************************************/

void RobotOpnCls( Mold_typ * pMold,Robot_OpnCls_Para_typ * pRobotOpnClsPara,Robot_OpnCls_Fix_typ * pRobotOpnClsFix);

/**************************************************************************************
     	        		I N I T U P  O F   T H E   T A S K
**************************************************************************************/
_INIT void init ( void )
{
	LMold.RobotOpnCls.Step = 0;
	RMold.RobotOpnCls.Step = 0;
} /* end of _INIT */

/*************************************************************************************
        				C Y C L I C   P A R T   O F   T H E   T A S K
**************************************************************************************/

_CYCLIC void cyclic ( void )
{

	if(LMold.TimeSet.RobotOpnAlarmTime == 0)LMold.TimeSet.RobotOpnAlarmTime= 1000;	/*  10s  */
	if(RMold.TimeSet.RobotOpnAlarmTime == 0)RMold.TimeSet.RobotOpnAlarmTime= 1000;	/*  10s  */

	if(LMold.TimeSet.RobotClsAlarmTime == 0)LMold.TimeSet.RobotClsAlarmTime= 1000;	/*  10s  */
	if(RMold.TimeSet.RobotClsAlarmTime == 0)RMold.TimeSet.RobotClsAlarmTime= 1000;	/*  10s  */

	LMold.TransDIn.RobotOpnLimit = ((0 == gMachineFix.MoldR.RobotOpnCls.bEnableRobotTwoOpnLimit && gMachineIn.LMold.RobotOpnLimit) ||
		( 1 == gMachineFix.MoldR.RobotOpnCls.bEnableRobotTwoOpnLimit &&  gMachineIn.LMold.RobotOpnLimitR && gMachineIn.LMold.RobotOpnLimitL));
	RMold.TransDIn.RobotOpnLimit = ((0 == gMachineFix.MoldR.RobotOpnCls.bEnableRobotTwoOpnLimit && gMachineIn.RMold.RobotOpnLimit) ||
		( 1 == gMachineFix.MoldR.RobotOpnCls.bEnableRobotTwoOpnLimit &&  gMachineIn.RMold.RobotOpnLimitR && gMachineIn.RMold.RobotOpnLimitL));

	//	LMold.TransDIn.RobotOpnLimitL = gMachineIn.LMold.RobotOpnLimitL;
	//	RMold.TransDIn.RobotOpnLimitL = gMachineIn.RMold.RobotOpnLimitL;
	//
	//	LMold.TransDIn.RobotOpnLimitR = gMachineIn.LMold.RobotOpnLimitR;
	//	RMold.TransDIn.RobotOpnLimitR = gMachineIn.RMold.RobotOpnLimitR;

	LMold.TransDIn.RobotClsLimit = gMachineIn.LMold.RobotClsLimit;
	RMold.TransDIn.RobotClsLimit = gMachineIn.RMold.RobotClsLimit;

	if(0 == gMachineFix.Option.bHideLeftStation)  // two mold
	{
		RobotOpnCls(&LMold,&gMachinePara.MoldL.RobotOpnCls,&gMachineFix.MoldL.RobotOpnCls);
	}
	RobotOpnCls(&RMold,&gMachinePara.MoldR.RobotOpnCls,&gMachineFix.MoldR.RobotOpnCls);

	gMachineOut.LMold.RobotCls = LMold.ValveOut.RobotCls;
	gMachineOut.RMold.RobotCls = RMold.ValveOut.RobotCls;

	gMachineOut.LMold.RobotOpn = LMold.ValveOut.RobotOpn;
	gMachineOut.RMold.RobotOpn = RMold.ValveOut.RobotOpn;

	/*-----------------------------------------------*/
	/*----------------- Robot OpnCls-----------------*/
	/*------------- ActuatorType--------------- */
	gMachineFix.MoldL.RobotOpnCls.eActuatorType = gMachineFix.MoldR.RobotOpnCls.eActuatorType;

	/*-------------- ValveType----------------- */
	gMachineFix.MoldL.RobotOpnCls.eValveType = gMachineFix.MoldR.RobotOpnCls.eValveType;

	/*------------ PressueOutputType--------------- */
	gMachineFix.MoldL.RobotOpnCls.ePressueOutputType = gMachineFix.MoldR.RobotOpnCls.ePressueOutputType;

	/*------------ FluxOutputType--------------- */
	gMachineFix.MoldL.RobotOpnCls.eFluxOutputType = gMachineFix.MoldR.RobotOpnCls.eFluxOutputType;

	/*------------ bEnableRobotClsLimit--------------- */
	gMachineFix.MoldL.RobotOpnCls.bEnableRobotClsLimit = gMachineFix.MoldR.RobotOpnCls.bEnableRobotClsLimit;

} /* end of _CYCLIC */

void RobotOpnCls( Mold_typ * pMold,Robot_OpnCls_Para_typ * pRobotOpnClsPara,Robot_OpnCls_Fix_typ * pRobotOpnClsFix)
{

	switch ( pMold->RobotOpnCls.Step )
	{
		/*------------------ stop all the output ------------------*/
		case 0:

			pMold->RobotOpnCls.Timer.IN = 0;
			pMold->RobotOpnCls.LimitTimer.IN   = 0;

			break;
		/*--------------------------------------------------- */
		/*------------------ Robot Close  ------------------- */
		/*--------------------------------------------------- */
		case 100:		/* cls delay */
			if(1 == pMold->Option.RobotOpnCls)
			{
				if(0 == pMold->RobotOpnCls.RobotFwTimeOutFlag)
				{
					if(pMold->TimeSet.RobotClsDly != 0)
					{
						pMold->RobotOpnCls.Timer.IN = 1;
						pMold->RobotOpnCls.Timer.PT = pMold->TimeSet.RobotClsDly;

						pMold->RobotOpnCls.Step = 200;
					}
					else
					{
						pMold->RobotOpnCls.Step = 300;
					}
				}
				else
				{
					pMold->RobotOpnCls.RobotFwTimeOutFlag = 0;
					pMold->RobotOpnCls.Step = 300;
				}

			}
			else
			{
				pMold->RobotOpnCls.Step = 300; // for no use
			}

			break;

		case 200:  		/* delay ok */
			pMold->TimeDis.RobotClsDly = pMold->RobotOpnCls.Timer.ET;
			if (1 == pMold->RobotOpnCls.Timer.Q)
			{
				pMold->RobotOpnCls.Timer.IN        = 0;
				pMold->RobotOpnCls.Step = 300;
			}
			break;

		case 300:  		/* set time */
			if( 1 == pMold->Option.RobotOpnCls)
			{
				pMold->RobotOpnCls.Timer.PT = pMold->TimeSet.RobotClsTime;
				pMold->RobotOpnCls.Timer.IN = 1;

				pMold->RobotOpnCls.LimitTimer.PT = pMold->TimeSet.RobotClsAlarmTime;
				pMold->RobotOpnCls.LimitTimer.IN = 1;

				pMold->RobotOpnCls.Step = 400;
			}
			else
			{
				pMold->RobotOpnCls.Step = 2900; // for no use
			}

			break;

		case 400:

			pMold->ActInfo.RobotOpn	= 0;
			pMold->ActInfo.RobotCls	= 1;

			switch (pRobotOpnClsFix->eActuatorType)
			{
				/*-------------------------------------------------*/
				case ACTUATOR_HYD: /*1:Oil*/
					/*-------------------------------------------------*/
					pMold->ValveOut.RobotOpn = 0;
					pMold->ValveOut.RobotCls = 1;

					pMold->RobotOpnCls.p_set = pRobotOpnClsPara->P_Cls;
					pMold->RobotOpnCls.v_set = pRobotOpnClsPara->V_Cls;

					if(1 == pMold->RobotOpnCls.Timer.Q)
					{
						pMold->ValveOut.RobotOpn = 0;
						pMold->ValveOut.RobotCls = 0;

						pMold->RobotOpnCls.p_set = 0;
						pMold->RobotOpnCls.v_set = 0;

						pMold->RobotOpnCls.Timer.IN = 0;
						pMold->RobotOpnCls.LimitTimer.IN   = 0;

						pMold->RobotOpnCls.Step = 500;
					}

					break;
				/*-------------------------------------------------*/
				case ACTUATOR_PNEU: /*2:Air*/
					/*-------------------------------------------------*/
					pMold->ValveOut.RobotOpn = 0;
					pMold->ValveOut.RobotCls = 1;

					if(0 == pRobotOpnClsFix->bEnableRobotClsLimit ||  1 == pMold->TransDIn.RobotClsLimit )
					{
						pMold->RobotOpnCls.Timer.IN = 0;
						pMold->RobotOpnCls.LimitTimer.IN   = 0;

						pMold->RobotOpnCls.Step = 500;
					}

					break;
			}

			break;

		case 500:
			switch (pRobotOpnClsFix->eActuatorType)
			{
				/*-------------------------------------------------*/
				case ACTUATOR_HYD: /*1:Oil*/
					/*-------------------------------------------------*/
					pMold->ActInfo.RobotOpn	= 0;
					pMold->ActInfo.RobotCls	= 0;

					pMold->ValveOut.RobotOpn = 0;
					pMold->ValveOut.RobotCls = 0;

					pMold->RobotOpnCls.p_set = 0;
					pMold->RobotOpnCls.v_set = 0;

					pMold->RobotOpnCls.Timer.IN = 0;
					pMold->RobotOpnCls.LimitTimer.IN   = 0;
					pMold->RobotOpnCls.Step = 3000;

					break;
				/*-------------------------------------------------*/
				case ACTUATOR_PNEU: /*2:Air*/
					/*-------------------------------------------------*/
					pMold->ActInfo.RobotOpn	= 0;
					pMold->ActInfo.RobotCls	= 1;

					pMold->ValveOut.RobotOpn = 0;
					pMold->ValveOut.RobotCls = 1;

					pMold->RobotOpnCls.Timer.IN = 0;
					pMold->RobotOpnCls.LimitTimer.IN   = 0;
					pMold->RobotOpnCls.Step = 3000;
					break;
			}

			break;

		case 2900:  // for no use

			pMold->ActInfo.RobotOpn	= 0;
			pMold->ActInfo.RobotCls	= 0;

			pMold->ValveOut.RobotOpn = 0;
			pMold->ValveOut.RobotCls = 0;

			pMold->RobotOpnCls.p_set = 0;
			pMold->RobotOpnCls.v_set = 0;

			pMold->RobotOpnCls.Timer.IN = 0;
			pMold->RobotOpnCls.LimitTimer.IN   = 0;
			pMold->RobotOpnCls.Step = 3000;

			break;

		case 3000:
			break;

		/* ---------------------- calibration Cls ---------------------- */
		case 5000:
			pMold->ActInfo.RobotOpn	= 0;
			pMold->ActInfo.RobotCls	= 1;

			pMold->ValveOut.RobotOpn = 0;
			pMold->ValveOut.RobotCls = 1;

			pMold->RobotOpnCls.p_set = pRobotOpnClsFix->pCalibCls;
			pMold->RobotOpnCls.v_set = pRobotOpnClsFix->vCalibCls;

			break;

		/*--------------------------------------------------- */
		/*------------------ Robot Open  -------------------- */
		/*--------------------------------------------------- */
		case 10100:		/* opn delay */
			if(1 == pMold->Option.RobotOpnCls)
			{
				switch (pRobotOpnClsFix->eActuatorType)
				{
					/*-------------------------------------------------*/
					case ACTUATOR_HYD: /*1:Oil*/
						/*-------------------------------------------------*/
						if(pMold->TimeSet.RobotOpnDly != 0)
						{
							pMold->RobotOpnCls.Timer.IN = 1;
							pMold->RobotOpnCls.Timer.PT = pMold->TimeSet.RobotOpnDly;

							pMold->RobotOpnCls.Step = 10200;
						}
						else
						{
							pMold->RobotOpnCls.Step = 10300;
						}

						break;
					/*-------------------------------------------------*/
					case ACTUATOR_PNEU: /*2:Air*/
						/*-------------------------------------------------*/
						if(pMold->TimeSet.RobotOpnDly != 0)
						{
							pMold->RobotOpnCls.Timer.IN = 1;
							pMold->RobotOpnCls.Timer.PT = pMold->TimeSet.RobotOpnDly;

							pMold->RobotOpnCls.Step = 10200;
						}
						else
						{
							pMold->RobotOpnCls.Step = 10300;
						}

						break;
				}
			}
			else
			{
				pMold->RobotOpnCls.Step = 10300;
			}

			break;

		case 10200:  		/* delay ok */
			pMold->TimeDis.RobotOpnDly = pMold->RobotOpnCls.Timer.ET;
			if (1 == pMold->RobotOpnCls.Timer.Q)
			{
				pMold->RobotOpnCls.Timer.IN  = 0;
				pMold->RobotOpnCls.Step = 10300;
			}
			break;

		case 10300:
			if(pMold->Option.RobotOpnCls)
			{
				pMold->RobotOpnCls.LimitTimer.IN = 1;
				pMold->RobotOpnCls.LimitTimer.PT = pMold->TimeSet.RobotOpnAlarmTime;
				pMold->RobotOpnCls.Step = 10400;
			}
			else  // for no use check limit
			{
				if (1 == pMold->TransDIn.RobotOpnLimit)
				{
					pMold->RobotOpnCls.Step = 12900;  // for no use
				}
				else
				{
					pMold->Alarm.RobotNotAtOpnPos = 1;
					pMold->RobotOpnCls.Step = 40000;           /*  Robot Open alarm   */
				}
			}

			break;

		case 10400:
			pMold->ActInfo.RobotOpn	= 1;
			pMold->ActInfo.RobotCls	= 0;

			pMold->ValveOut.RobotOpn = 1;
			pMold->ValveOut.RobotCls = 0;

			pMold->RobotOpnCls.p_set = pRobotOpnClsPara->P_Opn;
			pMold->RobotOpnCls.v_set = pRobotOpnClsPara->V_Opn;

			if (1 == pMold->TransDIn.RobotOpnLimit)
			{
				pMold->RobotOpnCls.p_set = 0;
				pMold->RobotOpnCls.v_set = 0;

				pMold->RobotOpnCls.Timer.IN = 0;
				pMold->RobotOpnCls.LimitTimer.IN   = 0;

				pMold->RobotOpnCls.Step = 10500;
			}
			break;

		case 10500: 			/* 夹时间 */

			if (1==gMachineInfo.Auto)
			{
				if(pMold == &RMold)
				{
					RMold.Option.RobotOpnCls = gMacOption.RRobotOpnCls;
				}
				else
				{
					LMold.Option.RobotOpnCls = gMacOption.LRobotOpnCls;
				}
			}

			pMold->ActInfo.RobotOpn	= 0;
			pMold->ActInfo.RobotCls	= 0;

			pMold->ValveOut.RobotOpn = 0;
			pMold->ValveOut.RobotCls = 0;

			pMold->RobotOpnCls.p_set = 0;
			pMold->RobotOpnCls.v_set = 0;

			pMold->RobotOpnCls.LimitTimer.IN = 0;
			pMold->RobotOpnCls.Timer.IN = 0;
			pMold->RobotOpnCls.Step = 13000;

			break;

		case 12900: //for no use
			pMold->ActInfo.RobotOpn	= 0;
			pMold->ActInfo.RobotCls	= 0;

			pMold->ValveOut.RobotOpn = 0;
			pMold->ValveOut.RobotCls = 0;

			pMold->RobotOpnCls.p_set = 0;
			pMold->RobotOpnCls.v_set = 0;

			pMold->RobotOpnCls.LimitTimer.IN = 0;
			pMold->RobotOpnCls.Timer.IN = 0;
			pMold->RobotOpnCls.Step = 13000;

			break;

		case 13000:
			break;

		/* ---------------------- calibration Opn ---------------------- */
		case 15000:
			pMold->ActInfo.RobotOpn	= 1;
			pMold->ActInfo.RobotCls	= 0;

			pMold->ValveOut.RobotOpn = 1;
			pMold->ValveOut.RobotCls = 0;

			pMold->RobotOpnCls.p_set = pRobotOpnClsFix->pCalibOpn;
			pMold->RobotOpnCls.v_set = pRobotOpnClsFix->vCalibOpn;

			break;

		/* ------------- Normal stop ------------- */
		case 20000:

//			pMold->ActInfo.RobotOpn	= 0;
//			pMold->ActInfo.RobotCls	= 0;
//
//			pMold->ValveOut.RobotOpn = 0;
//			pMold->ValveOut.RobotCls = 0;

			pMold->TimeDis.RobotClsDly 	= 0;
			pMold->TimeDis.RobotOpnDly 	= 0;

			pMold->RobotOpnCls.p_set = 0;
			pMold->RobotOpnCls.v_set = 0;

			pMold->RobotOpnCls.Timer.IN = 0;
			pMold->RobotOpnCls.LimitTimer.IN = 0;
			pMold->RobotOpnCls.Step = 0;

			break;

		/* ------------- Instancy stop ------------- */
		case 30000:
//			pMold->ActInfo.RobotOpn	= 0;
//			pMold->ActInfo.RobotCls	= 0;
//
//			pMold->ValveOut.RobotOpn = 0;
//			pMold->ValveOut.RobotCls = 0;

			pMold->RobotOpnCls.p_set = 0;
			pMold->RobotOpnCls.v_set = 0;

			pMold->RobotOpnCls.Timer.IN = 0;
			pMold->RobotOpnCls.LimitTimer.IN = 0;
			pMold->RobotOpnCls.Step = 0;

			break;

		/* ------------- Error stop ------------- */
		case 40000:
//			pMold->ActInfo.RobotOpn	= 0;
//			pMold->ActInfo.RobotCls	= 0;
//
//			pMold->ValveOut.RobotOpn = 0;
//			pMold->ValveOut.RobotCls = 0;

			pMold->RobotOpnCls.p_set = 0;
			pMold->RobotOpnCls.v_set = 0;

			pMold->RobotOpnCls.Timer.IN = 0;
			pMold->RobotOpnCls.LimitTimer.IN = 0;
			pMold->RobotOpnCls.Step = 0;

			break;

		/* ------------- auto run stop ------------- */
		case 41000:
//			pMold->ActInfo.RobotOpn	= 0;
//			pMold->ActInfo.RobotCls	= 0;
//
//			pMold->ValveOut.RobotOpn = 0;
//			pMold->ValveOut.RobotCls = 0;

			pMold->RobotOpnCls.Timer.IN = 0;
			pMold->RobotOpnCls.LimitTimer.IN = 0;
			pMold->RobotOpnCls.Step = 40000;

			break;
	}/* end of switch */

	/* ----------------- Robot Open / Close alarm time display --------------------  */
	if(pMold->RobotOpnCls.Step > 300 && pMold->RobotOpnCls.Step  < 500)			/* Robot Close  */
	{
		pMold->TimeDis.RobotClsAlarmTime = pMold->RobotOpnCls.LimitTimer.ET;
	}
	else if(pMold->RobotOpnCls.Step > 10300 && pMold->RobotOpnCls.Step  < 10500)	/* Robot Open   */
	{
		pMold->TimeDis.RobotOpnAlarmTime = pMold->RobotOpnCls.LimitTimer.ET;
	}

	/* ----------------- Robot Open / Close timeout --------------------  */
	if(1 == pMold->RobotOpnCls.LimitTimer.Q  && 1 == gMachineInfo.TimeLimit)
	{
		if(pMold->RobotOpnCls.Step < 3000 && pMold->RobotOpnCls.Step > 200)		/* Robot Close  */
		{
			pMold->Alarm.RobotNotAtClsPos = 1;
		}

		if(pMold->RobotOpnCls.Step < 13000 && pMold->RobotOpnCls.Step > 10200)	/* Robot Open   */
		{
			pMold->Alarm.RobotNotAtOpnPos = 1;
		}

		pMold->RobotOpnCls.Step = 41000;
	}/* if(1 == pMold->RobotOpnCls.LimitTimer.Q) */

	/* ----------------- Robot Open / Close action limit --------------------  */
	if(pMold->RobotOpnCls.Step < 3000 && pMold->RobotOpnCls.Step > 200)		/* Robot Close  */
	{

	}

	if(pMold->RobotOpnCls.Step < 13000 && pMold->RobotOpnCls.Step > 10200)	/* Robot Open   */
	{

	}

}/*end of function */
```

### Program Logical/process/chutedeflash (ANSIC, version 1.00.0) - chute deflash

#### chutedeflash.c
```c
/********************************************************************
 * COPYRIGHT --  B&R China
 ********************************************************************
 * Program: ChuteDeflashBlow
 * File: ChuteDeflashBlow.c
 * Author: lijianjun
 * Created: March 06, 2013
 ********************************************************************
 * Implementation of program ChuteDeflashBlow --- parison ChuteDeflashBlow control
 ********************************************************************/

#include <bur/plctypes.h>

#ifdef _DEFAULT_INCLUDES
#include <AsDefault.h>
#endif

/**************************************************************************************
                            Function Declarations
**************************************************************************************/

void ChuteDeflashBlow( Mold_typ * pMold);

/**************************************************************************************
     	        		I N I T U P  O F   T H E   T A S K
**************************************************************************************/
_INIT void init ( void )
 {
 	LMold.ChuteDeflashBlow.Step = 0;
 	RMold.ChuteDeflashBlow.Step = 0;
 } /* end of _INIT */

 /*************************************************************************************
        				C Y C L I C   P A R T   O F   T H E   T A S K
**************************************************************************************/

 _CYCLIC void cyclic ( void )
 {

	ChuteDeflashBlow(&LMold);
	ChuteDeflashBlow(&RMold);

	gMachineOut.LMold.ChuteDeflashBlow = LMold.ChuteDeflashBlow.Out;
	gMachineOut.RMold.ChuteDeflashBlow = RMold.ChuteDeflashBlow.Out;

 } /* end of _CYCLIC */

void ChuteDeflashBlow( Mold_typ * pMold)
{

	 switch ( pMold->ChuteDeflashBlow.Step )
    {
   		/*------------------ stop all the output ------------------*/
         case 0:
         	pMold->ChuteDeflashBlow.Out = 0;
         	pMold->ActInfo.ChuteDeflashBlow  = 0;
         	pMold->ChuteDeflashBlow.Timer.IN = 0;
         	break;

   		/*------------------ ChuteDeflashBlow  -------------------- */
   		case 100: 		/* ChuteDeflashBlow delay*/
  				if(pMold->TimeSet.ChuteDeflashBlowDelay != 0)
      		{
      			pMold->ChuteDeflashBlow.Timer.IN = 1;
  			      pMold->ChuteDeflashBlow.Timer.PT = pMold->TimeSet.ChuteDeflashBlowDelay;
      			pMold->ChuteDeflashBlow.Step = 200;
      		}
      		else
      		{
      			pMold->ChuteDeflashBlow.Step = 300;
      		}
       		break;
         case 200: 		/* ChuteDeflashBlow delay ok */
         	pMold->TimeDis.ChuteDeflashBlowDelay = pMold->ChuteDeflashBlow.Timer.ET;
         	if (1 == pMold->ChuteDeflashBlow.Timer.Q)
         	{
         		pMold->ChuteDeflashBlow.Timer.IN     = 0;
         		pMold->TimeDis.ChuteDeflashBlowDelay = 0;
         		pMold->ChuteDeflashBlow.Step = 300;
         	}
         	break;
         case 300:		/* ChuteDeflashBlow time */
         	if(pMold->TimeSet.ChuteDeflashBlowTime != 0)
         	{
         		pMold->ChuteDeflashBlow.Timer.IN = 1;
		         pMold->ChuteDeflashBlow.Timer.PT = pMold->TimeSet.ChuteDeflashBlowTime;
		         pMold->ChuteDeflashBlow.Step = 400;
         	}
         	else
         	{
         		pMold->ChuteDeflashBlow.Step = 500;
         	}
         	break;
         case 400:
         	pMold->ActInfo.ChuteDeflashBlow = 1;
         	pMold->ChuteDeflashBlow.Out     = 1;
         	pMold->TimeDis.ChuteDeflashBlowTime = pMold->ChuteDeflashBlow.Timer.ET;
         	if (1 == pMold->ChuteDeflashBlow.Timer.Q)
         	{
         		pMold->ChuteDeflashBlow.Out      = 0;
         		pMold->ChuteDeflashBlow.Timer.IN = 0;
         		pMold->TimeDis.ChuteDeflashBlowTime = 0;
         		pMold->ChuteDeflashBlow.Step = 500;
         	}
         	break;
         case 500:
         	pMold->ChuteDeflashBlow.Timer.IN = 0;
         	pMold->ChuteDeflashBlow.Out     = 0;
         	pMold->ActInfo.ChuteDeflashBlow = 0;
         	pMold->ChuteDeflashBlow.Step = 3000;
         	break;
         case 3000:
         	break;

         /* ------------- Normal stop ------------- */
         case 20000:
         	pMold->ChuteDeflashBlow.Out      = 0;
            pMold->ChuteDeflashBlow.Timer.IN = 0;

            pMold->ActInfo.ChuteDeflashBlow = 0;
            pMold->ChuteDeflashBlow.Step    = 0;
            break;

         /* ------------- Instance stop ------------- */
         case 30000:
         	pMold->ChuteDeflashBlow.Out      = 0;
         	pMold->ChuteDeflashBlow.Timer.IN = 0;

         	pMold->ActInfo.ChuteDeflashBlow  = 0;
         	pMold->ChuteDeflashBlow.Step     = 0;
         	break;

         /* ------------- Error stop ------------- */
         case 40000:
         	pMold->ChuteDeflashBlow.Out      = 0;
         	pMold->ChuteDeflashBlow.Timer.IN = 0;

         	pMold->ActInfo.ChuteDeflashBlow  = 0;
         	break;

	 }/* end of switch */
}/*end of function */
```

### Program Logical/process/screw (ANSIC, version 1.00.0) - screw

#### screw.c
```c
/********************************************************************
 * COPYRIGHT --  B&R China
 ********************************************************************
 * Program: screw
 * File: screw.c
 * Author: lijianjun
 * Created: March 06, 2013
 ********************************************************************
 * Implementation of program screw --- screw  up and down control
 ********************************************************************/

#include <bur/plctypes.h>

#ifdef _DEFAULT_INCLUDES
	#include <AsDefault.h>
#endif

/**************************************************************************************
                            Function Declarations
**************************************************************************************/

void Screw( Mold_typ * pMold,Screw_Para_typ * pScrewPara);

/**************************************************************************************
     	        		I N I T U P  O F   T H E   T A S K
**************************************************************************************/
_INIT void init ( void )
 {
 	LMold.Screw.Step = 30000;
 	RMold.Screw.Step = 30000;

 } /* end of _INIT */

 /*************************************************************************************
        				C Y C L I C   P A R T   O F   T H E   T A S K
**************************************************************************************/

 _CYCLIC void cyclic ( void )
 {
	RMold.TransDIn.ScrewFwLimit = gMachineIn.RMold.ScrewFwLimit;
	RMold.TransDIn.ScrewBwLimit = gMachineIn.RMold.ScrewBwLimit;

	LMold.TransDIn.ScrewFwLimit = gMachineIn.LMold.ScrewFwLimit;
	LMold.TransDIn.ScrewBwLimit = gMachineIn.LMold.ScrewBwLimit;

	if(!LMold.TimeSet.ScrewBwAlarmTime)LMold.TimeSet.ScrewBwAlarmTime = 500;  /* 5s  */
	if(!RMold.TimeSet.ScrewBwAlarmTime)RMold.TimeSet.ScrewBwAlarmTime = 500;  /* 5s  */

	if(!LMold.TimeSet.ScrewFwAlarmTime)LMold.TimeSet.ScrewFwAlarmTime = 500;  /* 5s  */
	if(!RMold.TimeSet.ScrewFwAlarmTime)RMold.TimeSet.ScrewFwAlarmTime = 500;  /* 5s  */

	Screw(&LMold,&gMachinePara.MoldL.Screw);
	Screw(&RMold,&gMachinePara.MoldR.Screw);

	gMachineOut.LMold.ScrewBw = LMold.ValveOut.ScrewBw;
	gMachineOut.LMold.ScrewFw = LMold.ValveOut.ScrewFw;

	gMachineOut.RMold.ScrewBw = RMold.ValveOut.ScrewBw;
	gMachineOut.RMold.ScrewFw = RMold.ValveOut.ScrewFw;

 } /* end of _CYCLIC */

void Screw( Mold_typ * pMold,Screw_Para_typ * pScrewPara)
{
	 switch ( pMold->Screw.Step )
    {
      	/*------------------ stop all the output ------------------*/
     	   case 0:
     		   pMold->ActInfo.ScrewFw  = 0;
     		   pMold->ActInfo.ScrewBw  = 0;
            pMold->Screw.Timer.IN	= 0;
            break;

        /*--------------- Screw forward -----------------*/
      	case 100: 	/* forward delay*/
      		if(1 == pMold->Option.Screw)
      		{
	      		pMold->Screw.Timer.IN = 1;
				   pMold->Screw.Timer.PT = pMold->TimeSet.ScrewFwDelay;
	      		pMold->Screw.Step = 200;
      		}
      	    else
      		{
      			pMold->Screw.Step = 3000;
      		}
            break;

         case 200: 	/* delay ok */
            pMold->TimeDis.ScrewFwDelay = pMold->Screw.Timer.ET;
            if (1 == pMold->Screw.Timer.Q)
            {
            	pMold->Screw.Timer.IN        = 0;
            	pMold->TimeDis.ScrewFwDelay = 0;
            	pMold->Screw.Step = 300;
            }
            break;

         case 300:
   			pMold->Screw.LimitTimer.IN = 1;
   			pMold->Screw.LimitTimer.PT = pMold->TimeSet.ScrewFwAlarmTime;
   			pMold->Screw.Step = 400;
            break;

         case 400:
            pMold->ActInfo.ScrewFw  = 1;
     		   pMold->ActInfo.ScrewBw  = 0;

			   pMold->ValveOut.ScrewFw = 1;
				pMold->ValveOut.ScrewBw = 0;

				pMold->Screw.p_set = pScrewPara->SpFw;
				pMold->Screw.v_set = pScrewPara->SvFw;

			   pMold->TimeDis.ScrewFwAlarmTime = pMold->Screw.LimitTimer.ET;

   			if(1 == pMold->TransDIn.ScrewFwLimit)
   			{
					pMold->Screw.p_set = 0;
					pMold->Screw.v_set = 0;

   				pMold->Screw.LimitTimer.IN = 0;
   				pMold->Screw.Step = 500;
   			}

   			if(1 == pMold->Screw.LimitTimer.Q)
   	        {
   				pMold->Screw.LimitTimer.IN = 0;
   				pMold->Alarm.ScrewNotAtFwPos = 1;
   				pMold->Screw.Step = 40000;
   			}
			   break;

		   case 500:
   			pMold->Screw.Timer.IN      = 0;
   			pMold->Screw.LimitTimer.IN = 0;

   			pMold->ActInfo.ScrewFw  = 0;
   			pMold->ValveOut.ScrewFw = 0;
   			pMold->Screw.Step = 3000;
   			break;

        case 3000:
            pMold->ActInfo.ScrewFw  = 0;
            break;

        /*------------------ Screw backward -------------------- */
     	  case 10100: 	/* Backward delay*/
      	   if(1 == pMold->Option.Screw)
      		{
      	      if(pMold->TimeSet.ScrewBwDelay != 0)
      			{
      				pMold->Screw.Timer.IN = 1;
					   pMold->Screw.Timer.PT = pMold->TimeSet.ScrewBwDelay;
      				pMold->Screw.Step 	= 10200;
      			}
      	      else
      			{
      				pMold->Screw.Step = 10300;
      			}
	      	}
      	  	else
      		{
      			pMold->Screw.Step = 13000;
      		}
            break;

       	case 10200: 	/* delay ok */
            pMold->TimeDis.ScrewBwDelay = pMold->Screw.Timer.ET;
            if (1 == pMold->Screw.Timer.Q)
            {
            	pMold->Screw.Timer.IN       = 0;
            	pMold->TimeDis.ScrewBwDelay = 0;
            	pMold->Screw.Step = 10300;
            }
            break;

       	case 10300:
			   pMold->Screw.LimitTimer.IN = 1;
            pMold->Screw.LimitTimer.PT = pMold->TimeSet.ScrewBwAlarmTime;
            pMold->Screw.Step = 10400;
			   break;

       	case 10400:
   			pMold->ActInfo.ScrewFw  = 0;
        		pMold->ActInfo.ScrewBw  = 1;

   			pMold->ValveOut.ScrewBw = 1;
   			pMold->ValveOut.ScrewFw = 0;

				pMold->Screw.p_set = pScrewPara->SpFw;
				pMold->Screw.v_set = pScrewPara->SvFw;

   			if(1 == pMold->TransDIn.ScrewBwLimit)
            {
					pMold->Screw.p_set = 0;
					pMold->Screw.v_set = 0;

               pMold->ActInfo.ScrewBw  = 0;
   				pMold->ValveOut.ScrewBw = 0;

   				pMold->Screw.Timer.IN = 0;
               pMold->Screw.Step = 10500;
            }

            pMold->TimeDis.ScrewBwAlarmTime = pMold->Screw.LimitTimer.ET;

            if(1 == pMold->Screw.LimitTimer.Q)
            {
            	pMold->Screw.Timer.IN   = 0;
            	pMold->Alarm.ScrewNotAtBwPos = 1;
            	pMold->Screw.Step = 40000;
            }
			   break;

		   case 10500:
   			pMold->ActInfo.ScrewFw  = 0;
        		pMold->ActInfo.ScrewBw  = 0;

   			pMold->ValveOut.ScrewBw = 0;

   			pMold->Screw.Timer.IN = 0;
   			pMold->Screw.LimitTimer.IN = 0;
   			pMold->Screw.Step = 13000;
   			break;

       	case 13000:
            break;

   		/*--------------- Manual action stop -----------------*/
           case 20000:
   			pMold->Screw.Timer.IN = 0;
   			pMold->Screw.LimitTimer.IN = 0;

   			pMold->ActInfo.ScrewFw = 0;
   			pMold->ActInfo.ScrewBw = 0;

   			pMold->ValveOut.ScrewFw = 0;
   			pMold->ValveOut.ScrewBw = 0;

				pMold->Screw.p_set = 0;
				pMold->Screw.v_set = 0;

   			pMold->Screw.Step = 0;
   			break;

   		/*--------------- Instancy stop -----------------*/
   		case 30000:
   			pMold->Screw.Timer.IN = 0;
   			pMold->Screw.LimitTimer.IN = 0;

   			pMold->ActInfo.ScrewFw = 0;
   			pMold->ActInfo.ScrewBw = 0;

   			pMold->ValveOut.ScrewFw = 0;
   			pMold->ValveOut.ScrewBw = 0;

				pMold->Screw.p_set = 0;
				pMold->Screw.v_set = 0;

   			pMold->Screw.Step = 0;
   			break;

   		/*--------------- Auto error stop -----------------*/
   		case 40000:
   			pMold->Screw.Timer.IN = 0;
   			pMold->Screw.LimitTimer.IN = 0;

   			pMold->ActInfo.ScrewFw = 0;
   			pMold->ActInfo.ScrewBw = 0;

   			pMold->ValveOut.ScrewFw = 0;
   			pMold->ValveOut.ScrewBw = 0;

				pMold->Screw.p_set = 0;
				pMold->Screw.v_set = 0;
   			break;
	}/* switch ( pMold->Screw.Step )  */
}
```

### Program Logical/process/pinpart (ANSIC, version 1.00.0) - pin part

#### pinpart.c
```c
/********************************************************************
 * COPYRIGHT --  B&R China
 ********************************************************************
 * Program: pinpart
 * File: pinpart.c
 * Author: lijianjun
 * Created: March 06, 2013
 ********************************************************************
 * Implementation of program pinpart --- pinpart control
 ********************************************************************/

#include <bur/plctypes.h>
#ifdef _DEFAULT_INCLUDES
	#include <AsDefault.h>
#endif

/**************************************************************************************
                            Function Declarations
**************************************************************************************/

void PinPart( Mold_typ * pMold);

/**************************************************************************************
     	        		I N I T U P  O F   T H E   T A S K
**************************************************************************************/
_INIT void init ( void )
 {
 	LMold.PinPart.Step = 30000;
 	RMold.PinPart.Step = 30000;

 } /* end of _INIT */

 /*************************************************************************************
        				C Y C L I C   P A R T   O F   T H E   T A S K
**************************************************************************************/

 _CYCLIC void cyclic ( void )
 {
	RMold.TransDIn.PinPartFwLimit = gMachineIn.RMold.PinPartFwLimit;
	RMold.TransDIn.PinPartBwLimit = gMachineIn.RMold.PinPartBwLimit;

	LMold.TransDIn.PinPartFwLimit = gMachineIn.LMold.PinPartFwLimit;
	LMold.TransDIn.PinPartBwLimit = gMachineIn.LMold.PinPartBwLimit;

	if(!LMold.TimeSet.PinPartBwAlarmTime)LMold.TimeSet.PinPartBwAlarmTime = 500;  /* 5s  */
	if(!RMold.TimeSet.PinPartBwAlarmTime)RMold.TimeSet.PinPartBwAlarmTime = 500;  /* 5s  */

	if(!LMold.TimeSet.PinPartFwAlarmTime)LMold.TimeSet.PinPartFwAlarmTime = 500;  /* 5s  */
	if(!RMold.TimeSet.PinPartFwAlarmTime)RMold.TimeSet.PinPartFwAlarmTime = 500;  /* 5s  */

	PinPart(&LMold);
	PinPart(&RMold);

	gMachineOut.LMold.PinPartBw = LMold.ValveOut.PinPartBw;
	gMachineOut.LMold.PinPartFw = LMold.ValveOut.PinPartFw;

	gMachineOut.RMold.PinPartBw = RMold.ValveOut.PinPartBw;
	gMachineOut.RMold.PinPartFw = RMold.ValveOut.PinPartFw;

 } /* end of _CYCLIC */

void PinPart( Mold_typ * pMold)
{

   switch ( pMold->PinPart.Step )
   {
      /*------------------ stop all the output ------------------*/
  	   case 0:
     		pMold->ActInfo.PinPartFw  = 0;
     		pMold->ActInfo.PinPartBw  = 0;
			pMold->ValveOut.PinPartFw = 0;
			pMold->ValveOut.PinPartBw = 0;

         pMold->PinPart.Out  		= 0;
         pMold->PinPart.Timer.IN	= 0;
         break;

     /*--------------- PinPart forward -----------------*/
   	case 100: 	/* forward delay*/
   		if(1 == pMold->Option.PinPart)
   		{
       		pMold->PinPart.Timer.IN = 1;
   	      pMold->PinPart.Timer.PT = pMold->TimeSet.PinPartFwDelay;
       		pMold->PinPart.Step = 200;
   		}
   	    else
   		{
   			pMold->PinPart.Step = 3000;
   		}
         break;

      case 200: 	/* delay ok */
         pMold->TimeDis.PinPartFwDelay = pMold->PinPart.Timer.ET;
         if (1 == pMold->PinPart.Timer.Q)
         {
         	pMold->PinPart.Timer.IN        = 0;
         	pMold->TimeDis.PinPartFwDelay = 0;
         	pMold->PinPart.Step = 300;
         }
         break;

      case 300:
			pMold->PinPart.LimitTimer.IN = 1;
			pMold->PinPart.LimitTimer.PT = pMold->TimeSet.PinPartFwAlarmTime;
			pMold->PinPart.Step = 400;
         break;

      case 400:
         pMold->ActInfo.PinPartFw  = 1;
     		pMold->ActInfo.PinPartBw  = 0;

			pMold->ValveOut.PinPartFw = 1;

			pMold->TimeDis.PinPartFwAlarmTime = pMold->PinPart.LimitTimer.ET;

			if(1 == pMold->TransDIn.PinPartFwLimit)
			{
				pMold->PinPart.LimitTimer.IN = 0;
				pMold->PinPart.Step = 500;
			}

			if(1 == pMold->PinPart.LimitTimer.Q)
	        {
				pMold->PinPart.LimitTimer.IN = 0;
				pMold->Alarm.PinPartNotAtFwPos = 1;
				pMold->PinPart.Step = 40000;
			}
         break;

      case 500:
			pMold->PinPart.Timer.IN      = 0;
			pMold->PinPart.LimitTimer.IN = 0;

			pMold->ActInfo.PinPartFw  = 0;
			pMold->ValveOut.PinPartFw = 0;
			pMold->PinPart.Step = 3000;
			break;

      case 3000:
         pMold->ActInfo.PinPartFw  = 0;
         break;

     /*------------------ PinPart backward -------------------- */
  	   case 10100: 	/* Backward delay*/
   	   if(1 == pMold->Option.PinPart)
   		{
   	      if(pMold->TimeSet.PinPartBwDelay != 0)
   			{
   				pMold->PinPart.Timer.IN = 1;
		         pMold->PinPart.Timer.PT = pMold->TimeSet.PinPartBwDelay;
   				pMold->PinPart.Step 	= 10200;
   			}
   	      else
   			{
   				pMold->PinPart.Step = 10300;
   			}
    	   }
   	  	else
   		{
   			pMold->PinPart.Step = 13000;
   		}
         break;

    	case 10200: 	/* delay ok */
         pMold->TimeDis.PinPartBwDelay = pMold->PinPart.Timer.ET;
         if (1 == pMold->PinPart.Timer.Q)
         {
         	pMold->PinPart.Timer.IN       = 0;
         	pMold->TimeDis.PinPartBwDelay = 0;
         	pMold->PinPart.Step = 10300;
         }
         break;

    	case 10300:
         pMold->PinPart.LimitTimer.IN = 1;
         pMold->PinPart.LimitTimer.PT = pMold->TimeSet.PinPartBwAlarmTime;
         pMold->PinPart.Step = 10400;
         break;

    	case 10400:
			pMold->ActInfo.PinPartFw  = 0;
     		pMold->ActInfo.PinPartBw  = 1;

			pMold->ValveOut.PinPartBw = 1;
			pMold->ValveOut.PinPartFw = 0;

			if(1 == pMold->TransDIn.PinPartBwLimit)
         {
            pMold->ActInfo.PinPartBw  = 0;
				pMold->ValveOut.PinPartBw = 0;

				pMold->PinPart.Timer.IN = 0;
            pMold->PinPart.Step = 10500;
         }

         pMold->TimeDis.PinPartBwAlarmTime = pMold->PinPart.LimitTimer.ET;

         if(1 == pMold->PinPart.LimitTimer.Q)
         {
         	pMold->PinPart.Timer.IN   = 0;
         	pMold->Alarm.PinPartNotAtBwPos = 1;
         	pMold->PinPart.Step = 40000;
         }
			break;

		case 10500:
			pMold->ActInfo.PinPartFw  = 0;
     		pMold->ActInfo.PinPartBw  = 0;

			pMold->ValveOut.PinPartBw = 0;

			pMold->PinPart.Timer.IN = 0;
			pMold->PinPart.LimitTimer.IN = 0;
			pMold->PinPart.Step = 13000;
			break;

      case 13000:
         break;

		case 18000:
			pMold->ActInfo.PinPartFw  = 0;
			pMold->ActInfo.PinPartBw  = 1;
			pMold->ValveOut.PinPartBw = 1;
			break;

		/*--------------- Manual action stop -----------------*/
      case 20000:
			pMold->PinPart.Timer.IN = 0;
			pMold->PinPart.LimitTimer.IN = 0;

			pMold->ActInfo.PinPartFw = 0;
			pMold->ActInfo.PinPartBw = 0;

			pMold->ValveOut.PinPartFw = 0;
			pMold->ValveOut.PinPartBw = 0;

			pMold->PinPart.Step = 0;
			break;

		/*--------------- Instancy stop -----------------*/
		case 30000:
			pMold->PinPart.Timer.IN = 0;
			pMold->PinPart.LimitTimer.IN = 0;

			pMold->ActInfo.PinPartFw = 0;
			pMold->ActInfo.PinPartBw = 0;

			pMold->ValveOut.PinPartFw = 0;
			pMold->ValveOut.PinPartBw = 0;

			pMold->PinPart.Step = 0;
			break;

		/*--------------- Auto error stop -----------------*/
		case 40000:
			pMold->PinPart.Timer.IN = 0;
			pMold->PinPart.LimitTimer.IN = 0;

			pMold->ActInfo.PinPartFw = 0;
			pMold->ActInfo.PinPartBw = 0;

			pMold->ValveOut.PinPartFw = 0;
			pMold->ValveOut.PinPartBw = 0;
			break;
	}/* switch ( pMold->PinPart.Step )  */
}/* end of function  */
```

### Program Logical/process/submold (ANSIC, version 1.00.0) - sub mold
